C01778=1014.459,160.454,-126.016,166.827,55.652,160.236
C01779=1014.455,160.205,-125.996,166.824,55.663,160.237
C01780=1014.451,159.957,-125.976,166.820,55.675,160.239
C01781=1014.447,159.707,-125.956,166.816,55.686,160.240
C01782=1014.443,159.458,-125.936,166.813,55.697,160.242
C01783=1014.439,159.209,-125.916,166.809,55.709,160.243
C01784=1014.435,158.960,-125.897,166.807,55.720,160.245
C01785=1014.431,158.710,-125.877,166.803,55.731,160.246
C01786=1014.428,158.461,-125.856,166.799,55.742,160.248
C01787=1014.423,158.212,-125.837,166.796,55.754,160.249
C01788=1014.419,157.963,-125.818,166.792,55.765,160.250
C01789=1014.415,157.714,-125.798,166.788,55.776,160.252
C01790=1014.411,157.464,-125.779,166.785,55.788,160.253
C01791=1014.406,157.215,-125.760,166.781,55.799,160.255
C01792=1014.403,156.966,-125.740,166.778,55.811,160.256
C01793=1014.398,156.716,-125.720,166.774,55.823,160.258
C01794=1014.393,156.467,-125.700,166.771,55.834,160.259
C01795=1014.389,156.217,-125.682,166.767,55.846,160.261
C01796=1014.385,155.968,-125.662,166.763,55.857,160.262
C01797=1014.381,155.719,-125.643,166.760,55.868,160.264
C01798=1014.376,155.470,-125.623,166.756,55.880,160.265
C01799=1014.372,155.221,-125.605,166.753,55.891,160.267
C01800=1014.367,154.941,-125.582,166.749,55.904,160.268
C01801=1014.363,154.661,-125.561,166.745,55.917,160.270
C01802=1014.358,154.381,-125.539,166.741,55.930,160.272
C01803=1014.354,154.101,-125.517,166.737,55.943,160.273
C01804=1014.350,153.852,-125.498,166.733,55.954,160.275
C01805=1014.345,153.602,-125.479,166.731,55.965,160.276
C01806=1014.341,153.353,-125.459,166.728,55.977,160.278
C01807=1014.337,153.104,-125.440,166.724,55.989,160.279
C01808=1014.333,152.855,-125.421,166.721,56.000,160.281
C01809=1014.328,152.606,-125.401,166.717,56.011,160.282
C01810=1014.324,152.356,-125.383,166.713,56.023,160.284
C01811=1014.320,152.108,-125.364,166.710,56.034,160.285
C01812=1014.316,151.858,-125.345,166.706,56.046,160.287
C01813=1014.312,151.609,-125.325,166.703,56.058,160.288
C01814=1014.308,151.360,-125.306,166.700,56.069,160.290
C01815=1014.304,151.110,-125.287,166.697,56.080,160.291
C01816=1014.299,150.861,-125.268,166.693,56.091,160.293
C01817=1014.295,150.612,-125.249,166.690,56.103,160.294
C01818=1014.291,150.363,-125.229,166.686,56.115,160.296
C01819=1014.287,150.113,-125.211,166.683,56.126,160.297
C01820=1014.283,149.864,-125.191,166.680,56.138,160.299
C01821=1014.279,149.615,-125.173,166.676,56.149,160.300
C01822=1014.275,149.366,-125.153,166.673,56.160,160.302
C01823=1014.270,149.116,-125.135,166.670,56.172,160.303
C01824=1014.266,148.867,-125.116,166.667,56.183,160.305
C01825=1014.262,148.618,-125.097,166.663,56.194,160.306
C01826=1014.257,148.369,-125.077,166.659,56.206,160.308
C01827=1014.253,148.119,-125.059,166.656,56.218,160.309
C01828=1014.249,147.870,-125.039,166.654,56.229,160.311
C01829=1014.245,147.621,-125.021,166.650,56.240,160.312
C01830=1014.241,147.372,-125.001,166.646,56.252,160.314
C01831=1014.237,147.122,-124.983,166.643,56.263,160.315
C01832=1014.233,146.873,-124.964,166.640,56.275,160.317
C01833=1014.229,146.624,-124.944,166.636,56.286,160.318
C01834=1014.224,146.374,-124.926,166.633,56.297,160.320
C01835=1014.220,146.126,-124.907,166.630,56.309,160.321
C01836=1014.216,145.876,-124.888,166.627,56.321,160.323
C01837=1014.212,145.627,-124.870,166.623,56.332,160.324
C01838=1014.208,145.378,-124.850,166.620,56.343,160.326
C01839=1014.204,145.128,-124.831,166.617,56.355,160.327
C01840=1014.199,144.879,-124.814,166.614,56.366,160.329
C01841=1014.195,144.630,-124.795,166.610,56.378,160.330
C01842=1014.191,144.381,-124.775,166.607,56.389,160.332
C01843=1014.186,144.131,-124.757,166.603,56.401,160.333
C01844=1014.182,143.882,-124.738,166.601,56.412,160.335
C01845=1014.178,143.633,-124.721,166.598,56.424,160.336
C01846=1014.174,143.384,-124.701,166.594,56.435,160.338
C01847=1014.170,143.134,-124.682,166.591,56.446,160.339
C01848=1014.165,142.885,-124.664,166.587,56.458,160.341
C01849=1014.161,142.636,-124.646,166.585,56.469,160.342
C01850=1014.157,142.386,-124.627,166.582,56.481,160.344
C01851=1014.153,142.137,-124.609,166.578,56.492,160.345
C01852=1014.148,141.888,-124.589,166.575,56.504,160.347
C01853=1014.145,141.639,-124.571,166.572,56.515,160.349
C01854=1014.140,141.390,-124.553,166.568,56.526,160.350
C01855=1014.136,141.140,-124.534,166.565,56.538,160.351
C01856=1014.132,140.890,-124.515,166.562,56.550,160.353
C01857=1014.128,140.642,-124.498,166.560,56.561,160.355
C01858=1014.124,140.392,-124.479,166.556,56.572,160.356
C01859=1014.119,140.143,-124.459,166.553,56.584,160.357
C01860=1014.115,139.894,-124.442,166.550,56.595,160.359
C01861=1014.111,139.645,-124.423,166.546,56.606,160.360
C01862=1014.107,139.395,-124.404,166.543,56.618,160.362
C01863=1014.102,139.146,-124.386,166.540,56.629,160.364
C01864=1014.098,138.866,-124.365,166.537,56.642,160.365
C01865=1014.094,138.586,-124.344,166.533,56.654,160.367
C01866=1014.088,138.306,-124.323,166.529,56.667,160.368
C01867=1014.085,138.026,-124.303,166.526,56.680,160.370
C01868=1014.080,137.776,-124.285,166.523,56.691,160.372
C01869=1014.076,137.527,-124.266,166.520,56.703,160.373
C01870=1014.072,137.278,-124.248,166.516,56.714,160.375
C01871=1014.068,137.028,-124.230,166.514,56.725,160.376
C01872=1014.063,136.779,-124.211,166.511,56.737,160.378
C01873=1014.060,136.530,-124.193,166.507,56.748,160.379
C01874=1014.055,136.281,-124.175,166.505,56.759,160.381
C01875=1014.051,136.031,-124.156,166.502,56.771,160.383
C01876=1014.047,135.782,-124.138,166.498,56.782,160.384
C01877=1014.043,135.533,-124.119,166.496,56.794,160.386
C01878=1014.038,135.283,-124.101,166.493,56.805,160.387
C01879=1014.034,135.034,-124.083,166.489,56.817,160.388
C01880=1014.030,134.784,-124.065,166.487,56.828,160.390
C01881=1014.025,134.535,-124.047,166.483,56.839,160.391
C01882=1014.022,134.286,-124.029,166.480,56.851,160.393
C01883=1014.017,134.037,-124.011,166.478,56.862,160.395
C01884=1014.013,133.788,-123.993,166.474,56.873,160.396
C01885=1014.009,133.538,-123.974,166.471,56.885,160.398
C01886=1014.004,133.288,-123.957,166.469,56.896,160.399
C01887=1014.001,133.039,-123.938,166.465,56.907,160.401
C01888=1013.996,132.790,-123.920,166.463,56.919,160.402
C01889=1013.992,132.541,-123.902,166.459,56.930,160.404
C01890=1013.988,132.291,-123.884,166.456,56.942,160.405
C01891=1013.984,132.043,-123.867,166.454,56.953,160.407
C01892=1013.979,131.793,-123.848,166.450,56.964,160.408
C01893=1013.975,131.544,-123.830,166.448,56.975,160.410
C01894=1013.971,131.295,-123.812,166.444,56.987,160.411
C01895=1013.967,131.045,-123.794,166.441,56.998,160.413
C01896=1013.963,130.796,-123.776,166.438,57.009,160.414
C01897=1013.958,130.547,-123.758,166.435,57.021,160.416
C01898=1013.955,130.298,-123.739,166.432,57.032,160.418
C01899=1013.950,130.048,-123.722,166.429,57.043,160.419
C01900=1013.946,129.798,-123.703,166.427,57.054,160.421
C01901=1013.942,129.549,-123.685,166.424,57.066,160.422
C01902=1013.938,129.299,-123.668,166.421,57.077,160.424
C01903=1013.933,129.051,-123.650,166.418,57.088,160.425
C01904=1013.929,128.801,-123.633,166.415,57.100,160.427
C01905=1013.925,128.552,-123.615,166.412,57.111,160.428
C01906=1013.921,128.302,-123.597,166.409,57.123,160.430
C01907=1013.917,128.053,-123.579,166.406,57.135,160.431
C01908=1013.912,127.803,-123.562,166.403,57.145,160.433
C01909=1013.908,127.555,-123.544,166.400,57.157,160.435
C01910=1013.904,127.305,-123.526,166.397,57.168,160.436
C01911=1013.899,127.056,-123.509,166.394,57.180,160.438
C01912=1013.895,126.806,-123.491,166.391,57.192,160.439
C01913=1013.891,126.557,-123.474,166.389,57.202,160.441
C01914=1013.886,126.307,-123.456,166.386,57.214,160.442
C01915=1013.882,126.058,-123.439,166.383,57.225,160.444
C01916=1013.878,125.809,-123.421,166.380,57.237,160.445
C01917=1013.874,125.559,-123.404,166.377,57.247,160.447
C01918=1013.869,125.310,-123.386,166.374,57.259,160.448
C01919=1013.865,125.061,-123.368,166.371,57.270,160.450
C01920=1013.861,124.811,-123.351,166.369,57.282,160.452
C01921=1013.856,124.562,-123.333,166.366,57.294,160.453
C01922=1013.852,124.312,-123.316,166.363,57.304,160.455
C01923=1013.848,124.064,-123.298,166.360,57.316,160.456
C01924=1013.843,123.814,-123.281,166.357,57.327,160.458
C01925=1013.839,123.564,-123.263,166.354,57.338,160.459
C01926=1013.835,123.315,-123.245,166.352,57.350,160.461
C01927=1013.831,123.066,-123.228,166.348,57.361,160.462
C01928=1013.826,122.786,-123.209,166.346,57.373,160.464
C01929=1013.821,122.506,-123.189,166.342,57.386,160.466
C01930=1013.817,122.226,-123.169,166.340,57.399,160.468
C01931=1013.812,121.946,-123.150,166.336,57.411,160.469
C01932=1013.807,121.697,-123.132,166.334,57.423,160.471
C01933=1013.803,121.447,-123.115,166.330,57.434,160.472
C01934=1013.799,121.197,-123.097,166.328,57.445,160.474
C01935=1013.795,120.949,-123.080,166.326,57.456,160.475
C01936=1013.791,120.699,-123.063,166.322,57.467,160.477
C01937=1013.786,120.449,-123.045,166.319,57.478,160.478
C01938=1013.782,120.201,-123.027,166.316,57.490,160.480
C01939=1013.778,119.952,-123.010,166.314,57.501,160.481
C01940=1013.774,119.702,-122.993,166.311,57.511,160.483
C01941=1013.770,119.453,-122.975,166.308,57.523,160.485
C01942=1013.765,119.203,-122.958,166.306,57.534,160.486
C01943=1013.761,118.954,-122.940,166.302,57.545,160.487
C01944=1013.757,118.704,-122.923,166.300,57.557,160.489
C01945=1013.753,118.455,-122.905,166.298,57.568,160.491
C01946=1013.749,118.206,-122.888,166.294,57.579,160.492
C01947=1013.745,117.956,-122.871,166.292,57.589,160.493
C01948=1013.740,117.707,-122.854,166.290,57.601,160.495
C01949=1013.736,117.458,-122.836,166.286,57.612,160.497
C01950=1013.732,117.209,-122.819,166.284,57.623,160.498
C01951=1013.728,116.959,-122.801,166.281,57.634,160.500
C01952=1013.724,116.709,-122.784,166.279,57.645,160.501
C01953=1013.720,116.461,-122.766,166.276,57.656,160.503
C01954=1013.715,116.211,-122.749,166.273,57.667,160.504
C01955=1013.712,115.961,-122.731,166.271,57.678,160.506
C01956=1013.708,115.712,-122.714,166.267,57.689,160.507
C01957=1013.704,115.462,-122.697,166.265,57.700,160.509
C01958=1013.700,115.213,-122.679,166.263,57.711,160.510
C01959=1013.696,114.964,-122.662,166.261,57.722,160.512
C01960=1013.691,114.714,-122.644,166.257,57.733,160.513
C01961=1013.687,114.465,-122.627,166.255,57.744,160.515
C01962=1013.683,114.215,-122.610,166.252,57.755,160.516
C01963=1013.680,113.966,-122.593,166.250,57.766,160.518
C01964=1013.675,113.717,-122.575,166.247,57.777,160.519
C01965=1013.671,113.468,-122.558,166.244,57.788,160.521
C01966=1013.667,113.218,-122.541,166.241,57.799,160.522
C01967=1013.663,112.969,-122.524,166.239,57.809,160.524
C01968=1013.659,112.719,-122.506,166.237,57.821,160.526
C01969=1013.655,112.470,-122.489,166.235,57.832,160.527
C01970=1013.651,112.221,-122.472,166.232,57.843,160.529
C01971=1013.647,111.972,-122.454,166.229,57.854,160.530
C01972=1013.642,111.722,-122.437,166.226,57.865,160.532
C01973=1013.638,111.473,-122.421,166.224,57.875,160.533
C01974=1013.634,111.224,-122.403,166.221,57.886,160.535
C01975=1013.630,110.973,-122.387,166.218,57.897,160.536
C01976=1013.625,110.724,-122.370,166.215,57.908,160.537
C01977=1013.621,110.475,-122.353,166.213,57.919,160.539
C01978=1013.617,110.226,-122.336,166.211,57.930,160.541
C01979=1013.613,109.977,-122.320,166.208,57.941,160.542
C01980=1013.608,109.727,-122.302,166.205,57.953,160.544
C01981=1013.604,109.477,-122.285,166.203,57.964,160.545
C01982=1013.600,109.228,-122.268,166.201,57.974,160.547
C01983=1013.596,108.979,-122.251,166.198,57.985,160.548
C01984=1013.591,108.729,-122.234,166.196,57.996,160.550
C01985=1013.587,108.480,-122.218,166.192,58.007,160.551
C01986=1013.583,108.230,-122.201,166.190,58.018,160.553
C01987=1013.579,107.981,-122.185,166.188,58.029,160.554
C01988=1013.575,107.732,-122.168,166.185,58.040,160.556
C01989=1013.570,107.482,-122.151,166.183,58.051,160.557
C01990=1013.566,107.233,-122.134,166.179,58.062,160.559
C01991=1013.561,106.984,-122.118,166.177,58.073,160.560
C01992=1013.557,106.704,-122.099,166.175,58.085,160.562
C01993=1013.552,106.423,-122.081,166.172,58.097,160.564
C01994=1013.547,106.144,-122.061,166.169,58.109,160.566
C01995=1013.542,105.864,-122.043,166.166,58.121,160.567
C01996=1013.538,105.615,-122.026,166.163,58.133,160.569
C01997=1013.534,105.365,-122.010,166.161,58.144,160.570
C01998=1013.530,105.116,-121.993,166.158,58.154,160.572
C01999=1013.525,104.867,-121.976,166.156,58.165,160.573
C02000=1013.522,104.617,-121.960,166.154,58.176,160.575
C02001=1013.517,104.367,-121.943,166.151,58.187,160.576
C02002=1013.513,104.118,-121.926,166.149,58.198,160.578
C02003=1013.508,103.869,-121.910,166.147,58.209,160.579
C02004=1013.505,103.619,-121.893,166.144,58.220,160.581
C02005=1013.500,103.370,-121.877,166.141,58.231,160.582
C02006=1013.496,103.121,-121.860,166.139,58.242,160.584
C02007=1013.492,102.871,-121.844,166.136,58.253,160.586
C02008=1013.488,102.622,-121.827,166.133,58.263,160.587
C02009=1013.483,102.372,-121.811,166.131,58.274,160.588
C02010=1013.479,102.123,-121.794,166.129,58.285,160.590
C02011=1013.475,101.874,-121.777,166.126,58.295,160.591
C02012=1013.471,101.624,-121.761,166.124,58.306,160.593
C02013=1013.467,101.374,-121.744,166.122,58.317,160.595
C02014=1013.463,101.125,-121.727,166.119,58.327,160.596
C02015=1013.459,100.876,-121.711,166.117,58.338,160.597
C02016=1013.454,100.627,-121.694,166.114,58.349,160.599
C02017=1013.450,100.377,-121.677,166.112,58.360,160.601
C02018=1013.446,100.128,-121.662,166.109,58.370,160.602
C02019=1013.442,99.878,-121.644,166.107,58.381,160.603
C02020=1013.437,99.628,-121.628,166.106,58.391,160.605
C02021=1013.434,99.379,-121.611,166.103,58.402,160.607
C02022=1013.429,99.130,-121.595,166.100,58.412,160.608
C02023=1013.425,98.880,-121.578,166.098,58.423,160.610
C02024=1013.421,98.631,-121.562,166.096,58.434,160.611
C02025=1013.416,98.382,-121.546,166.093,58.444,160.612
C02026=1013.412,98.132,-121.530,166.091,58.455,160.614
C02027=1013.408,97.883,-121.513,166.088,58.466,160.616
C02028=1013.404,97.633,-121.498,166.086,58.477,160.617
C02029=1013.399,97.384,-121.481,166.084,58.488,160.619
C02030=1013.395,97.135,-121.465,166.081,58.498,160.620
C02031=1013.391,96.885,-121.449,166.079,58.509,160.622
C02032=1013.387,96.636,-121.432,166.077,58.520,160.623
C02033=1013.383,96.386,-121.417,166.074,58.530,160.624
C02034=1013.378,96.137,-121.401,166.072,58.541,160.626
C02035=1013.374,95.888,-121.384,166.069,58.552,160.628
C02036=1013.370,95.638,-121.368,166.067,58.563,160.629
C02037=1013.366,95.388,-121.352,166.064,58.573,160.630
C02038=1013.361,95.139,-121.336,166.062,58.584,160.632
C02039=1013.357,94.890,-121.320,166.059,58.594,160.633
C02040=1013.353,94.640,-121.304,166.058,58.605,160.635
C02041=1013.349,94.391,-121.287,166.056,58.616,160.637
C02042=1013.344,94.141,-121.271,166.053,58.626,160.638
C02043=1013.340,93.892,-121.256,166.051,58.637,160.639
C02044=1013.335,93.643,-121.239,166.048,58.647,160.641
C02045=1013.331,93.393,-121.223,166.046,58.658,160.642
C02046=1013.328,93.143,-121.207,166.043,58.669,160.644
C02047=1013.323,92.894,-121.191,166.042,58.679,160.645
C02048=1013.319,92.645,-121.175,166.040,58.689,160.647
C02049=1013.314,92.395,-121.159,166.037,58.700,160.648
C02050=1013.310,92.146,-121.143,166.035,58.711,160.650
C02051=1013.306,91.896,-121.126,166.032,58.721,160.651
C02052=1013.302,91.647,-121.110,166.031,58.731,160.653
C02053=1013.298,91.397,-121.095,166.028,58.742,160.654
C02054=1013.293,91.148,-121.078,166.025,58.752,160.655
C02055=1013.289,90.899,-121.062,166.023,58.763,160.657
C02056=1013.285,90.619,-121.044,166.021,58.774,160.659
C02057=1013.279,90.339,-121.026,166.018,58.786,160.660
C02058=1013.275,90.060,-121.008,166.015,58.798,160.662
C02059=1013.270,89.781,-120.990,166.013,58.809,160.664
C02060=1013.266,89.531,-120.975,166.011,58.819,160.665
C02061=1013.262,89.282,-120.958,166.008,58.830,160.667
C02062=1013.258,89.032,-120.942,166.007,58.840,160.668
C02063=1013.254,88.782,-120.927,166.004,58.850,160.669
C02064=1013.249,88.533,-120.910,166.002,58.861,160.671
C02065=1013.245,88.284,-120.894,166.000,58.871,160.673
C02066=1013.240,88.034,-120.879,165.998,58.882,160.674
C02067=1013.236,87.785,-120.863,165.995,58.892,160.675
C02068=1013.232,87.535,-120.847,165.992,58.902,160.677
C02069=1013.227,87.286,-120.831,165.991,58.913,160.679
C02070=1013.223,87.036,-120.816,165.989,58.923,160.680
C02071=1013.219,86.787,-120.800,165.986,58.934,160.681
C02072=1013.214,86.538,-120.785,165.984,58.944,160.683
C02073=1013.210,86.288,-120.769,165.982,58.954,160.684
C02074=1013.206,86.039,-120.753,165.980,58.965,160.686
C02075=1013.201,85.789,-120.738,165.977,58.975,160.687
C02076=1013.197,85.539,-120.722,165.975,58.985,160.689
C02077=1013.193,85.290,-120.706,165.973,58.996,160.690
C02078=1013.189,85.040,-120.691,165.971,59.006,160.692
C02079=1013.185,84.790,-120.675,165.969,59.016,160.693
C02080=1013.180,84.542,-120.660,165.966,59.026,160.694
C02081=1013.176,84.292,-120.645,165.964,59.037,160.696
C02082=1013.172,84.042,-120.629,165.962,59.047,160.697
C02083=1013.167,83.793,-120.613,165.960,59.057,160.699
C02084=1013.163,83.543,-120.597,165.958,59.067,160.700
C02085=1013.159,83.294,-120.582,165.955,59.077,160.702
C02086=1013.154,83.044,-120.566,165.954,59.087,160.703
C02087=1013.151,82.795,-120.550,165.952,59.098,160.705
C02088=1013.146,82.546,-120.535,165.949,59.108,160.706
C02089=1013.141,82.296,-120.520,165.947,59.118,160.708
C02090=1013.137,82.047,-120.504,165.945,59.128,160.709
C02091=1013.133,81.797,-120.488,165.943,59.138,160.710
C02092=1013.129,81.548,-120.473,165.940,59.149,160.712
C02093=1013.125,81.298,-120.458,165.939,59.158,160.713
C02094=1013.121,81.049,-120.442,165.936,59.169,160.714
C02095=1013.116,80.799,-120.426,165.934,59.178,160.716
C02096=1013.111,80.550,-120.411,165.932,59.189,160.717
C02097=1013.107,80.300,-120.395,165.930,59.199,160.719
C02098=1013.103,80.051,-120.380,165.927,59.209,160.720
C02099=1013.099,79.802,-120.364,165.926,59.219,160.722
C02100=1013.095,79.551,-120.349,165.923,59.229,160.723
C02101=1013.091,79.302,-120.333,165.921,59.239,160.724
C02102=1013.086,79.052,-120.317,165.920,59.249,160.726
C02103=1013.083,78.803,-120.302,165.917,59.259,160.727
C02104=1013.078,78.554,-120.287,165.915,59.269,160.729
C02105=1013.073,78.305,-120.271,165.913,59.279,160.730
C02106=1013.069,78.055,-120.255,165.911,59.289,160.732
C02107=1013.066,77.806,-120.240,165.910,59.299,160.733
C02108=1013.061,77.556,-120.225,165.906,59.308,160.734
C02109=1013.057,77.306,-120.209,165.905,59.318,160.736
C02110=1013.053,77.057,-120.193,165.903,59.328,160.737
C02111=1013.049,76.807,-120.178,165.900,59.338,160.739
C02112=1013.044,76.558,-120.163,165.899,59.348,160.740
C02113=1013.040,76.308,-120.148,165.897,59.358,160.742
C02114=1013.036,76.059,-120.132,165.894,59.367,160.743
C02115=1013.031,75.809,-120.117,165.892,59.377,160.744
C02116=1013.027,75.560,-120.102,165.891,59.387,160.746
C02117=1013.023,75.311,-120.086,165.888,59.397,160.747
C02118=1013.018,75.061,-120.072,165.887,59.407,160.749
C02119=1013.014,74.811,-120.056,165.884,59.418,160.750
C02120=1013.010,74.572,-120.042,165.882,59.427,160.751
C02121=1013.006,74.331,-120.027,165.880,59.436,160.752
C02122=1013.002,74.092,-120.013,165.878,59.446,160.754
C02123=1012.997,73.852,-119.998,165.876,59.455,160.755
C02124=1012.994,73.612,-119.983,165.874,59.465,160.757
C02125=1012.989,73.372,-119.969,165.872,59.474,160.758
C02126=1012.985,73.133,-119.955,165.870,59.484,160.759
C02127=1012.981,72.892,-119.940,165.868,59.493,160.761
C02128=1012.977,72.643,-119.925,165.867,59.503,160.762
C02129=1012.973,72.393,-119.910,165.865,59.512,160.763
C02130=1012.968,72.144,-119.895,165.862,59.522,160.765
C02131=1012.964,71.895,-119.879,165.860,59.532,160.766
C02132=1012.959,71.645,-119.865,165.858,59.541,160.767
C02133=1012.955,71.396,-119.849,165.857,59.551,160.769
C02134=1012.951,71.147,-119.835,165.854,59.560,160.770
C02135=1012.947,70.897,-119.819,165.852,59.570,160.771
C02136=1012.943,70.647,-119.804,165.850,59.580,160.773
C02137=1012.938,70.398,-119.789,165.848,59.589,160.774
C02138=1012.934,70.148,-119.774,165.847,59.599,160.776
C02139=1012.929,69.899,-119.759,165.844,59.608,160.777
C02140=1012.926,69.649,-119.744,165.843,59.618,160.779
C02141=1012.921,69.400,-119.729,165.840,59.628,160.780
C02142=1012.917,69.150,-119.714,165.838,59.638,160.781
C02143=1012.912,68.901,-119.699,165.836,59.647,160.782
C02144=1012.908,68.651,-119.684,165.835,59.657,160.784
C02145=1012.903,68.402,-119.669,165.832,59.666,160.785
C02146=1012.900,68.152,-119.654,165.830,59.675,160.786
C02147=1012.895,67.903,-119.639,165.829,59.685,160.788
C02148=1012.891,67.653,-119.624,165.827,59.694,160.789
C02149=1012.887,67.404,-119.610,165.825,59.704,160.791
C02150=1012.882,67.154,-119.594,165.823,59.713,160.792
C02151=1012.878,66.904,-119.580,165.821,59.723,160.793
C02152=1012.874,66.655,-119.565,165.818,59.733,160.794
C02153=1012.869,66.405,-119.550,165.816,59.742,160.796
C02154=1012.865,66.156,-119.536,165.815,59.752,160.797
C02155=1012.861,65.906,-119.521,165.812,59.761,160.798
C02156=1012.856,65.657,-119.506,165.810,59.770,160.800
C02157=1012.853,65.407,-119.491,165.809,59.780,160.801
C02158=1012.848,65.157,-119.477,165.807,59.789,160.802
C02159=1012.843,64.909,-119.462,165.805,59.798,160.804
C02160=1012.839,64.659,-119.447,165.803,59.808,160.805
C02161=1012.835,64.409,-119.432,165.801,59.817,160.806
C02162=1012.830,64.160,-119.417,165.799,59.826,160.808
C02163=1012.826,63.910,-119.402,165.797,59.836,160.809
C02164=1012.822,63.661,-119.388,165.795,59.845,160.811
C02165=1012.817,63.411,-119.374,165.793,59.855,160.812
C02166=1012.813,63.161,-119.358,165.791,59.864,160.813
C02167=1012.809,62.912,-119.344,165.790,59.873,160.814
C02168=1012.804,62.662,-119.329,165.788,59.882,160.816
C02169=1012.801,62.413,-119.315,165.786,59.891,160.817
C02170=1012.796,62.163,-119.300,165.784,59.901,160.818
C02171=1012.791,61.913,-119.286,165.782,59.910,160.820
C02172=1012.787,61.664,-119.272,165.780,59.919,160.821
C02173=1012.782,61.414,-119.257,165.778,59.928,160.822
C02174=1012.778,61.165,-119.243,165.777,59.938,160.824
C02175=1012.773,60.915,-119.228,165.775,59.947,160.825
C02176=1012.769,60.666,-119.214,165.773,59.957,160.826
C02177=1012.764,60.416,-119.200,165.770,59.966,160.827
C02178=1012.760,60.167,-119.185,165.768,59.975,160.829
C02179=1012.755,59.917,-119.171,165.766,59.984,160.830
C02180=1012.732,71.816,-120.285,165.827,59.747,160.800
C02181=1012.736,72.066,-120.299,165.829,59.737,160.799
C02182=1012.741,72.316,-120.315,165.831,59.728,160.797
C02183=1012.745,72.565,-120.329,165.833,59.719,160.796
C02184=1012.749,72.814,-120.345,165.834,59.709,160.795
C02185=1012.753,73.059,-120.359,165.837,59.700,160.793
C02186=1012.757,73.305,-120.373,165.839,59.691,160.792
C02187=1012.762,73.551,-120.388,165.840,59.681,160.791
C02188=1012.765,73.796,-120.403,165.842,59.672,160.789
C02189=1012.770,74.042,-120.418,165.844,59.662,160.788
C02190=1012.774,74.286,-120.433,165.846,59.653,160.787
C02191=1012.778,74.532,-120.448,165.848,59.644,160.785
C02192=1012.783,74.778,-120.463,165.851,59.633,160.784
C02193=1012.787,75.026,-120.478,165.853,59.624,160.783
C02194=1012.791,75.276,-120.493,165.854,59.614,160.781
C02195=1012.796,75.526,-120.508,165.856,59.604,160.780
C02196=1012.799,75.775,-120.523,165.858,59.595,160.778
C02197=1012.803,76.025,-120.539,165.861,59.585,160.777
C02198=1012.809,76.274,-120.554,165.863,59.576,160.776
C02199=1012.812,76.524,-120.569,165.864,59.566,160.774
C02200=1012.816,76.773,-120.584,165.866,59.556,160.773
C02201=1012.820,77.024,-120.599,165.868,59.547,160.772
C02202=1012.825,77.273,-120.615,165.871,59.537,160.770
C02203=1012.829,77.522,-120.630,165.873,59.528,160.769
C02204=1012.833,77.771,-120.646,165.874,59.518,160.767
C02205=1012.837,78.021,-120.661,165.876,59.508,160.766
C02206=1012.842,78.271,-120.677,165.879,59.498,160.765
C02207=1012.845,78.520,-120.692,165.881,59.488,160.763
C02208=1012.850,78.769,-120.708,165.882,59.478,160.762
C02209=1012.854,79.020,-120.723,165.884,59.469,160.761
C02210=1012.858,79.268,-120.738,165.887,59.459,160.759
C02211=1012.862,79.518,-120.753,165.889,59.449,160.758
C02212=1012.867,79.767,-120.769,165.890,59.439,160.756
C02213=1012.871,80.017,-120.785,165.894,59.430,160.755
C02214=1012.874,80.266,-120.800,165.895,59.420,160.754
C02215=1012.879,80.516,-120.815,165.897,59.410,160.752
C02216=1012.883,80.766,-120.831,165.899,59.400,160.751
C02217=1012.887,81.015,-120.847,165.901,59.390,160.749
C02218=1012.891,81.264,-120.862,165.902,59.380,160.748
C02219=1012.896,81.513,-120.878,165.906,59.371,160.747
C02220=1012.900,81.764,-120.893,165.907,59.361,160.745
C02221=1012.904,82.013,-120.908,165.910,59.350,160.744
C02222=1012.908,82.262,-120.924,165.911,59.341,160.742
C02223=1012.912,82.512,-120.940,165.913,59.331,160.741
C02224=1012.917,82.761,-120.955,165.916,59.320,160.740
C02225=1012.921,83.011,-120.971,165.917,59.311,160.738
C02226=1012.925,83.261,-120.986,165.920,59.300,160.737
C02227=1012.929,83.509,-121.001,165.922,59.290,160.735
C02228=1012.934,83.759,-121.017,165.924,59.280,160.734
C02229=1012.938,84.009,-121.032,165.926,59.270,160.732
C02230=1012.942,84.258,-121.048,165.928,59.260,160.731
C02231=1012.947,84.508,-121.064,165.930,59.250,160.729
C02232=1012.950,84.757,-121.079,165.933,59.240,160.728
C02233=1012.954,85.007,-121.094,165.934,59.230,160.727
C02234=1012.959,85.256,-121.110,165.937,59.220,160.725
C02235=1012.964,85.506,-121.125,165.939,59.210,160.724
C02236=1012.968,85.755,-121.141,165.941,59.200,160.722
C02237=1012.972,86.005,-121.157,165.942,59.189,160.721
C02238=1012.976,86.254,-121.172,165.945,59.179,160.719
C02239=1012.980,86.503,-121.188,165.948,59.169,160.718
C02240=1012.985,86.753,-121.204,165.949,59.159,160.716
C02241=1012.989,87.002,-121.220,165.952,59.149,160.715
C02242=1012.993,87.252,-121.235,165.954,59.139,160.714
C02243=1012.997,87.502,-121.251,165.956,59.128,160.712
C02244=1013.002,87.750,-121.266,165.958,59.117,160.711
C02245=1013.006,88.000,-121.282,165.960,59.108,160.709
C02246=1013.010,88.250,-121.297,165.963,59.097,160.708
C02247=1013.015,88.500,-121.313,165.965,59.086,160.706
C02248=1013.019,88.749,-121.328,165.966,59.077,160.705
C02249=1013.023,88.998,-121.345,165.969,59.066,160.703
C02250=1013.027,89.248,-121.361,165.972,59.056,160.702
C02251=1013.031,89.498,-121.377,165.974,59.046,160.701
C02252=1013.035,89.746,-121.392,165.976,59.035,160.699
C02253=1013.041,90.026,-121.410,165.978,59.024,160.697
C02254=1013.045,90.306,-121.429,165.981,59.013,160.696
C02255=1013.049,90.585,-121.446,165.982,59.001,160.694
C02256=1013.054,90.864,-121.464,165.986,58.990,160.693
C02257=1013.058,91.114,-121.480,165.988,58.979,160.691
C02258=1013.062,91.363,-121.496,165.989,58.969,160.689
C02259=1013.067,91.613,-121.512,165.992,58.959,160.688
C02260=1013.070,91.862,-121.529,165.995,58.948,160.687
C02261=1013.075,92.112,-121.545,165.996,58.938,160.685
C02262=1013.078,92.360,-121.560,165.999,58.928,160.684
C02263=1013.083,92.610,-121.576,166.001,58.917,160.682
C02264=1013.087,92.860,-121.592,166.004,58.906,160.681
C02265=1013.091,93.109,-121.609,166.005,58.897,160.679
C02266=1013.095,93.358,-121.624,166.008,58.886,160.678
C02267=1013.100,93.608,-121.640,166.010,58.876,160.676
C02268=1013.104,93.858,-121.656,166.013,58.865,160.675
C02269=1013.108,94.107,-121.672,166.014,58.855,160.673
C02270=1013.112,94.356,-121.689,166.017,58.845,160.672
C02271=1013.116,94.606,-121.705,166.019,58.834,160.670
C02272=1013.121,94.856,-121.720,166.022,58.823,160.669
C02273=1013.125,95.105,-121.737,166.024,58.812,160.668
C02274=1013.130,95.354,-121.753,166.026,58.803,160.666
C02275=1013.133,95.604,-121.769,166.028,58.792,160.664
C02276=1013.137,95.854,-121.785,166.030,58.781,160.663
C02277=1013.142,96.103,-121.801,166.033,58.771,160.662
C02278=1013.146,96.352,-121.817,166.035,58.760,160.660
C02279=1013.151,96.602,-121.833,166.038,58.749,160.659
C02280=1013.154,96.850,-121.849,166.040,58.739,160.657
C02281=1013.158,97.100,-121.865,166.042,58.729,160.656
C02282=1013.163,97.349,-121.881,166.044,58.718,160.654
C02283=1013.167,97.599,-121.897,166.047,58.708,160.653
C02284=1013.171,97.848,-121.913,166.049,58.697,160.651
C02285=1013.175,98.098,-121.930,166.051,58.686,160.650
C02286=1013.179,98.347,-121.945,166.054,58.675,160.648
C02287=1013.184,98.596,-121.962,166.056,58.665,160.647
C02288=1013.187,98.846,-121.978,166.058,58.654,160.645
C02289=1013.193,99.096,-121.995,166.061,58.643,160.644
C02290=1013.196,99.346,-122.011,166.063,58.632,160.642
C02291=1013.201,99.595,-122.028,166.066,58.622,160.641
C02292=1013.204,99.845,-122.044,166.067,58.612,160.639
C02293=1013.209,100.094,-122.061,166.069,58.601,160.638
C02294=1013.213,100.344,-122.077,166.072,58.591,160.636
C02295=1013.217,100.592,-122.094,166.074,58.580,160.635
C02296=1013.221,100.842,-122.110,166.077,58.570,160.633
C02297=1013.225,101.091,-122.126,166.079,58.559,160.632
C02298=1013.229,101.341,-122.143,166.082,58.548,160.630
C02299=1013.234,101.590,-122.159,166.084,58.537,160.629
C02300=1013.237,101.839,-122.176,166.087,58.527,160.627
C02301=1013.242,102.089,-122.192,166.089,58.516,160.626
C02302=1013.246,102.338,-122.209,166.091,58.505,160.624
C02303=1013.250,102.588,-122.225,166.094,58.495,160.623
C02304=1013.254,102.837,-122.242,166.096,58.484,160.621
C02305=1013.258,103.087,-122.258,166.099,58.473,160.620
C02306=1013.262,103.336,-122.275,166.101,58.462,160.618
C02307=1013.267,103.585,-122.291,166.104,58.452,160.617
C02308=1013.270,103.835,-122.308,166.106,58.441,160.615
C02309=1013.275,104.084,-122.324,166.108,58.430,160.614
C02310=1013.278,104.334,-122.341,166.111,58.419,160.612
C02311=1013.284,104.583,-122.357,166.113,58.408,160.611
C02312=1013.287,104.833,-122.375,166.115,58.397,160.609
C02313=1013.292,105.082,-122.390,166.118,58.387,160.608
C02314=1013.296,105.331,-122.407,166.120,58.376,160.606
C02315=1013.300,105.580,-122.424,166.123,58.365,160.605
C02316=1013.304,105.830,-122.440,166.125,58.355,160.603
C02317=1013.309,106.110,-122.460,166.129,58.342,160.602
C02318=1013.314,106.390,-122.478,166.131,58.330,160.600
C02319=1013.318,106.669,-122.496,166.133,58.317,160.598
C02320=1013.323,106.949,-122.514,166.136,58.305,160.596
C02321=1013.327,107.198,-122.531,166.138,58.294,160.595
C02322=1013.332,107.447,-122.548,166.141,58.283,160.593
C02323=1013.335,107.697,-122.564,166.143,58.273,160.592
C02324=1013.340,107.947,-122.582,166.146,58.261,160.590
C02325=1013.344,108.196,-122.598,166.149,58.250,160.589
C02326=1013.348,108.446,-122.615,166.151,58.240,160.587
C02327=1013.352,108.695,-122.631,166.153,58.229,160.585
C02328=1013.356,108.944,-122.648,166.156,58.218,160.584
C02329=1013.361,109.193,-122.665,166.158,58.207,160.582
C02330=1013.364,109.443,-122.681,166.161,58.196,160.581
C02331=1013.369,109.693,-122.698,166.164,58.185,160.579
C02332=1013.374,109.942,-122.715,166.166,58.174,160.578
C02333=1013.377,110.191,-122.732,166.168,58.163,160.576
C02334=1013.381,110.440,-122.749,166.171,58.152,160.575
C02335=1013.385,110.690,-122.766,166.174,58.141,160.573
C02336=1013.390,110.939,-122.782,166.177,58.130,160.572
C02337=1013.394,111.189,-122.799,166.179,58.119,160.570
C02338=1013.398,111.439,-122.816,166.181,58.108,160.569
C02339=1013.402,111.688,-122.833,166.184,58.098,160.567
C02340=1013.406,111.937,-122.850,166.187,58.086,160.566
C02341=1013.410,112.186,-122.867,166.189,58.075,160.564
C02342=1013.415,112.436,-122.885,166.192,58.065,160.563
C02343=1013.419,112.685,-122.902,166.194,58.054,160.561
C02344=1013.422,112.935,-122.919,166.196,58.043,160.560
C02345=1013.426,113.184,-122.936,166.199,58.032,160.558
C02346=1013.430,113.433,-122.953,166.202,58.021,160.557
C02347=1013.435,113.683,-122.970,166.205,58.010,160.555
C02348=1013.439,113.932,-122.988,166.207,57.999,160.554
C02349=1013.443,114.181,-123.005,166.209,57.988,160.552
C02350=1013.447,114.430,-123.022,166.212,57.977,160.551
C02351=1013.451,114.680,-123.040,166.215,57.966,160.549
C02352=1013.455,114.930,-123.057,166.218,57.955,160.548
C02353=1013.459,115.179,-123.074,166.220,57.945,160.546
C02354=1013.463,115.428,-123.091,166.222,57.934,160.545
C02355=1013.467,115.678,-123.108,166.226,57.923,160.543
C02356=1013.471,115.927,-123.125,166.228,57.911,160.541
C02357=1013.475,116.176,-123.143,166.230,57.900,160.540
C02358=1013.479,116.425,-123.160,166.233,57.889,160.538
C02359=1013.484,116.675,-123.178,166.236,57.878,160.537
C02360=1013.487,116.924,-123.195,166.238,57.867,160.536
C02361=1013.491,117.174,-123.212,166.241,57.857,160.534
C02362=1013.495,117.423,-123.229,166.243,57.846,160.532
C02363=1013.500,117.673,-123.246,166.246,57.834,160.531
C02364=1013.504,117.922,-123.264,166.249,57.823,160.529
C02365=1013.508,118.171,-123.281,166.251,57.812,160.528
C02366=1013.511,118.421,-123.299,166.255,57.801,160.526
C02367=1013.515,118.670,-123.316,166.256,57.789,160.525
C02368=1013.519,118.920,-123.334,166.260,57.778,160.523
C02369=1013.523,119.168,-123.351,166.262,57.767,160.522
C02370=1013.528,119.418,-123.369,166.265,57.757,160.520
C02371=1013.532,119.668,-123.386,166.268,57.745,160.519
C02372=1013.536,119.917,-123.403,166.270,57.734,160.517
C02373=1013.540,120.167,-123.420,166.273,57.723,160.516
C02374=1013.544,120.415,-123.438,166.276,57.712,160.514
C02375=1013.548,120.665,-123.455,166.278,57.700,160.512
C02376=1013.553,120.915,-123.473,166.282,57.689,160.511
C02377=1013.556,121.164,-123.490,166.284,57.678,160.510
C02378=1013.561,121.413,-123.508,166.287,57.666,160.508
C02379=1013.565,121.663,-123.525,166.290,57.656,160.506
C02380=1013.569,121.912,-123.542,166.291,57.644,160.505
C02381=1013.574,122.191,-123.561,166.295,57.632,160.503
C02382=1013.578,122.471,-123.581,166.298,57.619,160.501
C02383=1013.584,122.752,-123.600,166.302,57.607,160.500
C02384=1013.588,123.032,-123.620,166.305,57.594,160.498
C02385=1013.592,123.280,-123.638,166.307,57.582,160.496
C02386=1013.597,123.530,-123.655,166.311,57.571,160.495
C02387=1013.600,123.780,-123.673,166.313,57.560,160.493
C02388=1013.605,124.028,-123.690,166.316,57.548,160.492
C02389=1013.609,124.278,-123.708,166.319,57.538,160.490
C02390=1013.613,124.527,-123.725,166.322,57.526,160.489
C02391=1013.617,124.777,-123.742,166.324,57.515,160.487
C02392=1013.622,125.026,-123.760,166.327,57.503,160.485
C02393=1013.626,125.275,-123.777,166.330,57.492,160.484
C02394=1013.630,125.525,-123.795,166.333,57.480,160.482
C02395=1013.634,125.774,-123.812,166.335,57.470,160.481
C02396=1013.639,126.024,-123.830,166.338,57.458,160.479
C02397=1013.643,126.273,-123.848,166.342,57.447,160.478
C02398=1013.647,126.522,-123.865,166.344,57.435,160.476
C02399=1013.651,126.772,-123.882,166.347,57.423,160.474
C02400=1013.655,127.020,-123.900,166.349,57.412,160.473
C02401=1013.660,127.270,-123.917,166.352,57.401,160.471
C02402=1013.664,127.520,-123.934,166.356,57.389,160.470
C02403=1013.668,127.769,-123.953,166.358,57.378,160.468
C02404=1013.672,128.018,-123.970,166.361,57.366,160.467
C02405=1013.677,128.268,-123.988,166.365,57.355,160.465
C02406=1013.681,128.517,-124.005,166.367,57.343,160.464
C02407=1013.685,128.766,-124.022,166.370,57.332,160.462
C02408=1013.690,129.016,-124.040,166.373,57.320,160.461
C02409=1013.694,129.265,-124.057,166.375,57.309,160.459
C02410=1013.698,129.515,-124.076,166.379,57.298,160.458
C02411=1013.702,129.765,-124.093,166.381,57.286,160.456
C02412=1013.705,130.013,-124.112,166.384,57.275,160.454
C02413=1013.710,130.263,-124.130,166.388,57.263,160.453
C02414=1013.714,130.512,-124.147,166.390,57.253,160.451
C02415=1013.718,130.762,-124.166,166.393,57.241,160.450
C02416=1013.722,131.010,-124.184,166.396,57.230,160.448
C02417=1013.727,131.260,-124.201,166.399,57.218,160.447
C02418=1013.730,131.509,-124.219,166.403,57.207,160.445
C02419=1013.735,131.759,-124.238,166.405,57.196,160.444
C02420=1013.738,132.008,-124.255,166.408,57.185,160.442
C02421=1013.743,132.258,-124.273,166.410,57.173,160.440
C02422=1013.747,132.506,-124.291,166.413,57.161,160.439
C02423=1013.751,132.756,-124.310,166.417,57.150,160.438
C02424=1013.755,133.005,-124.327,166.419,57.139,160.436
C02425=1013.760,133.255,-124.345,166.423,57.128,160.435
C02426=1013.763,133.503,-124.364,166.426,57.116,160.433
C02427=1013.768,133.753,-124.381,166.428,57.104,160.431
C02428=1013.771,134.002,-124.400,166.432,57.093,160.430
C02429=1013.776,134.252,-124.418,166.435,57.081,160.428
C02430=1013.780,134.500,-124.435,166.437,57.070,160.427
C02431=1013.784,134.751,-124.454,166.440,57.059,160.425
C02432=1013.789,135.000,-124.472,166.444,57.047,160.424
C02433=1013.792,135.249,-124.490,166.447,57.035,160.422
C02434=1013.797,135.498,-124.508,166.449,57.025,160.421
C02435=1013.800,135.747,-124.527,166.453,57.013,160.419
C02436=1013.805,135.997,-124.544,166.456,57.001,160.417
C02437=1013.809,136.246,-124.562,166.458,56.990,160.416
C02438=1013.813,136.496,-124.581,166.461,56.979,160.414
C02439=1013.818,136.745,-124.599,166.465,56.967,160.413
C02440=1013.821,136.994,-124.617,166.468,56.956,160.411
C02441=1013.826,137.243,-124.635,166.470,56.944,160.410
C02442=1013.829,137.492,-124.654,166.474,56.932,160.408
C02443=1013.834,137.742,-124.671,166.477,56.921,160.407
C02444=1013.838,137.992,-124.690,166.481,56.910,160.405
C02445=1013.843,138.271,-124.711,166.483,56.897,160.403
C02446=1013.847,138.551,-124.732,166.487,56.884,160.402
C02447=1013.851,138.831,-124.752,166.490,56.871,160.400
C02448=1013.857,139.111,-124.773,166.494,56.858,160.398
C02449=1013.861,139.361,-124.792,166.497,56.848,160.397
C02450=1013.864,139.609,-124.810,166.500,56.836,160.395
C02451=1013.869,139.859,-124.828,166.503,56.824,160.394
C02452=1013.872,140.108,-124.847,166.506,56.812,160.392
C02453=1013.876,140.357,-124.865,166.509,56.802,160.391
C02454=1013.881,140.607,-124.884,166.512,56.790,160.389
C02455=1013.885,140.856,-124.902,166.516,56.778,160.388
C02456=1013.889,141.105,-124.920,166.519,56.767,160.386
C02457=1013.893,141.355,-124.939,166.522,56.755,160.385
C02458=1013.897,141.604,-124.957,166.525,56.744,160.383
C02459=1013.902,141.853,-124.975,166.528,56.732,160.381
C02460=1013.906,142.103,-124.994,166.532,56.721,160.380
C02461=1013.909,142.352,-125.013,166.535,56.709,160.379
C02462=1013.914,142.601,-125.031,166.538,56.698,160.377
C02463=1013.918,142.850,-125.050,166.540,56.686,160.375
C02464=1013.922,143.100,-125.069,166.544,56.674,160.374
C02465=1013.926,143.348,-125.087,166.547,56.663,160.372
C02466=1013.930,143.598,-125.106,166.551,56.652,160.371
C02467=1013.934,143.848,-125.124,166.554,56.640,160.369
C02468=1013.939,144.096,-125.142,166.557,56.628,160.368
C02469=1013.943,144.346,-125.161,166.560,56.616,160.366
C02470=1013.947,144.596,-125.180,166.564,56.605,160.365
C02471=1013.952,144.844,-125.198,166.566,56.594,160.363
C02472=1013.955,145.093,-125.217,166.570,56.582,160.362
C02473=1013.959,145.343,-125.236,166.573,56.571,160.360
C02474=1013.963,145.593,-125.254,166.576,56.559,160.358
C02475=1013.968,145.841,-125.273,166.580,56.548,160.357
C02476=1013.972,146.090,-125.292,166.583,56.536,160.356
C02477=1013.976,146.340,-125.310,166.587,56.524,160.354
C02478=1013.980,146.590,-125.329,166.589,56.513,160.352
C02479=1013.984,146.839,-125.349,166.592,56.501,160.351
C02480=1013.988,147.088,-125.367,166.596,56.490,160.350
C02481=1013.992,147.337,-125.386,166.599,56.479,160.348
C02482=1013.997,147.586,-125.405,166.603,56.467,160.346
C02483=1014.001,147.836,-125.423,166.606,56.455,160.345
C02484=1014.005,148.085,-125.442,166.609,56.444,160.343
C02485=1014.009,148.334,-125.461,166.612,56.432,160.342
C02486=1014.013,148.583,-125.480,166.615,56.421,160.340
C02487=1014.017,148.833,-125.499,166.619,56.410,160.339
C02488=1014.021,149.082,-125.518,166.622,56.398,160.337
C02489=1014.025,149.332,-125.537,166.625,56.386,160.336
C02490=1014.029,149.580,-125.556,166.629,56.374,160.334
C02491=1014.033,149.830,-125.575,166.632,56.364,160.333
C02492=1014.037,150.079,-125.594,166.636,56.352,160.331
C02493=1014.041,150.329,-125.613,166.639,56.340,160.330
C02494=1014.046,150.578,-125.633,166.642,56.328,160.328
C02495=1014.050,150.827,-125.651,166.646,56.317,160.327
C02496=1014.054,151.075,-125.670,166.649,56.305,160.325
C02497=1014.058,151.325,-125.689,166.652,56.293,160.324
C02498=1014.063,151.574,-125.708,166.656,56.282,160.322
C02499=1014.067,151.824,-125.727,166.660,56.271,160.321
C02500=1014.071,152.073,-125.746,166.663,56.259,160.319
C02501=1014.075,152.322,-125.765,166.666,56.247,160.318
C02502=1014.079,152.571,-125.785,166.670,56.236,160.316
C02503=1014.083,152.820,-125.803,166.673,56.224,160.315
C02504=1014.087,153.069,-125.822,166.676,56.212,160.313
C02505=1014.091,153.319,-125.841,166.679,56.201,160.311
C02506=1014.095,153.568,-125.861,166.682,56.189,160.310
C02507=1014.099,153.817,-125.881,166.686,56.179,160.309
C02508=1014.103,154.067,-125.899,166.689,56.167,160.307
C02509=1014.108,154.347,-125.922,166.694,56.154,160.306
C02510=1014.113,154.627,-125.943,166.698,56.140,160.304
C02511=1014.118,154.907,-125.964,166.702,56.127,160.302
C02512=1014.122,155.187,-125.986,166.706,56.115,160.301
C02513=1014.126,155.436,-126.005,166.709,56.103,160.299
C02514=1014.131,155.685,-126.025,166.712,56.091,160.297
C02515=1014.134,155.934,-126.043,166.716,56.080,160.296
C02516=1014.139,156.183,-126.063,166.719,56.068,160.294
C02517=1014.143,156.432,-126.082,166.723,56.056,160.293
C02518=1014.146,156.682,-126.101,166.726,56.045,160.291
C02519=1014.151,156.931,-126.121,166.729,56.033,160.290
C02520=1014.155,157.180,-126.140,166.733,56.021,160.288
C02521=1014.159,157.429,-126.160,166.736,56.010,160.287
C02522=1014.163,157.679,-126.179,166.740,55.998,160.285
C02523=1014.168,157.928,-126.198,166.743,55.987,160.284
C02524=1014.172,158.177,-126.218,166.747,55.976,160.282
C02525=1014.176,158.426,-126.238,166.751,55.964,160.281
C02526=1014.180,158.675,-126.257,166.754,55.952,160.279
C02527=1014.184,158.925,-126.277,166.757,55.941,160.278
C02528=1014.187,159.174,-126.297,166.761,55.929,160.276
C02529=1014.192,159.423,-126.317,166.765,55.918,160.275
C02530=1014.195,159.672,-126.337,166.768,55.907,160.274
C02531=1014.200,159.921,-126.356,166.772,55.895,160.272
C02532=1014.203,160.171,-126.376,166.775,55.884,160.271
C02533=1014.208,160.420,-126.396,166.779,55.873,160.269
C02534=1014.211,160.669,-126.416,166.783,55.861,160.268
C02535=1014.215,160.918,-126.436,166.786,55.849,160.266
C02536=1014.219,161.168,-126.455,166.790,55.838,160.265
C02537=1014.223,161.417,-126.475,166.794,55.827,160.264
C02538=1014.227,161.666,-126.495,166.797,55.815,160.262
C02539=1014.231,161.915,-126.515,166.801,55.804,160.261
C02540=1014.235,162.164,-126.534,166.804,55.792,160.259
C02541=1014.240,162.414,-126.556,166.808,55.781,160.257
C02542=1014.243,162.663,-126.576,166.811,55.769,160.256
C02543=1014.247,162.912,-126.595,166.815,55.758,160.255
C02544=1014.251,163.162,-126.615,166.819,55.747,160.253
C02545=1014.255,163.411,-126.635,166.822,55.735,160.252
C02546=1014.259,163.660,-126.655,166.826,55.723,160.250
C02547=1014.264,163.908,-126.675,166.829,55.712,160.249
C02548=1014.267,164.158,-126.695,166.833,55.700,160.247
C02549=1014.271,164.407,-126.715,166.837,55.689,160.246
C02550=1014.275,164.656,-126.735,166.840,55.678,160.244
C02551=1014.279,164.905,-126.755,166.845,55.666,160.243
C02552=1014.283,165.154,-126.774,166.848,55.654,160.242
C02553=1014.287,165.403,-126.795,166.852,55.643,160.240
C02554=1014.292,165.653,-126.815,166.855,55.631,160.239
C02555=1014.296,165.902,-126.835,166.859,55.620,160.237
C02556=1014.299,166.152,-126.855,166.863,55.608,160.236
C02557=1014.304,166.400,-126.875,166.866,55.597,160.234
C02558=1014.308,166.649,-126.895,166.870,55.586,160.233
C02559=1014.312,166.898,-126.915,166.874,55.574,160.231
C02560=1014.316,167.148,-126.935,166.878,55.562,160.230
C02561=1014.319,167.397,-126.955,166.882,55.551,160.228
C02562=1014.324,167.646,-126.975,166.885,55.539,160.227
C02563=1014.328,167.896,-126.995,166.889,55.528,160.225
C02564=1014.333,168.144,-127.016,166.893,55.516,160.224
C02565=1014.336,168.393,-127.036,166.896,55.505,160.222
C02566=1014.341,168.642,-127.055,166.901,55.493,160.221
C02567=1014.345,168.892,-127.076,166.904,55.481,160.220
C02568=1014.349,169.141,-127.096,166.908,55.470,160.218
C02569=1014.353,169.390,-127.116,166.912,55.458,160.217
C02570=1014.357,169.639,-127.137,166.915,55.447,160.215
C02571=1014.361,169.888,-127.156,166.920,55.435,160.214
C02572=1014.366,170.138,-127.176,166.923,55.423,160.212
C02573=1014.370,170.418,-127.199,166.927,55.411,160.211
C02574=1014.375,170.697,-127.222,166.933,55.397,160.209
C02575=1014.379,170.976,-127.245,166.936,55.384,160.207
C02576=1014.384,171.256,-127.267,166.940,55.372,160.206
C02577=1014.388,171.505,-127.287,166.945,55.360,160.204
C02578=1014.393,171.755,-127.308,166.949,55.348,160.203
C02579=1014.397,172.004,-127.328,166.952,55.337,160.201
C02580=1014.401,172.253,-127.348,166.956,55.325,160.200
C02581=1014.405,172.502,-127.368,166.960,55.313,160.199
C02582=1014.409,172.751,-127.389,166.964,55.302,160.197
C02583=1014.414,173.000,-127.408,166.968,55.290,160.196
C02584=1014.417,173.249,-127.429,166.972,55.278,160.194
C02585=1014.422,173.499,-127.450,166.976,55.267,160.193
C02586=1014.426,173.748,-127.469,166.980,55.255,160.191
C02587=1014.430,173.997,-127.490,166.984,55.244,160.190
C02588=1014.435,174.246,-127.510,166.988,55.232,160.188
C02589=1014.439,174.495,-127.531,166.992,55.221,160.187
C02590=1014.443,174.744,-127.550,166.996,55.209,160.186
C02591=1014.447,174.993,-127.571,167.000,55.197,160.184
C02592=1014.452,175.243,-127.591,167.003,55.185,160.182
C02593=1014.456,175.491,-127.611,167.008,55.173,160.181
C02594=1014.461,175.741,-127.633,167.011,55.162,160.180
C02595=1014.465,175.990,-127.652,167.015,55.150,160.178
C02596=1014.469,176.239,-127.673,167.020,55.138,160.177
C02597=1014.473,176.489,-127.693,167.024,55.127,160.175
C02598=1014.478,176.737,-127.713,167.028,55.115,160.174
C02599=1014.481,176.986,-127.734,167.032,55.104,160.173
C02600=1014.487,177.236,-127.754,167.036,55.092,160.171
C02601=1014.491,177.484,-127.775,167.040,55.080,160.170
C02602=1014.495,177.734,-127.795,167.044,55.069,160.168
C02603=1014.499,177.983,-127.815,167.049,55.057,160.167
C02604=1014.503,178.232,-127.836,167.052,55.045,160.165
C02605=1014.508,178.481,-127.856,167.056,55.034,160.164
C02606=1014.512,178.730,-127.877,167.060,55.022,160.162
C02607=1014.516,178.980,-127.897,167.064,55.010,160.161
C02608=1014.521,179.228,-127.918,167.069,54.998,160.160
C02609=1014.526,179.478,-127.939,167.073,54.987,160.158
C02610=1014.530,179.726,-127.959,167.077,54.975,160.157
C02611=1014.534,179.976,-127.979,167.081,54.964,160.155
C02612=1014.538,180.225,-128.000,167.085,54.951,160.154
C02613=1014.543,180.474,-128.020,167.089,54.940,160.152
C02614=1014.547,180.724,-128.041,167.094,54.928,160.151
C02615=1014.552,180.972,-128.061,167.097,54.917,160.149
C02616=1014.556,181.221,-128.082,167.102,54.905,160.148
C02617=1014.560,181.470,-128.103,167.106,54.893,160.147
C02618=1014.565,181.720,-128.123,167.111,54.882,160.145
C02619=1014.569,181.969,-128.144,167.114,54.870,160.144
C02620=1014.573,182.218,-128.166,167.118,54.859,160.142
C02621=1014.577,182.468,-128.188,167.122,54.847,160.141
C02622=1014.581,182.716,-128.208,167.127,54.836,160.140
C02623=1014.585,182.965,-128.229,167.131,54.825,160.138
C02624=1014.589,183.215,-128.251,167.135,54.814,160.137
C02625=1014.593,183.463,-128.272,167.140,54.802,160.135
C02626=1014.597,183.713,-128.293,167.143,54.790,160.134
C02627=1014.601,183.962,-128.314,167.147,54.779,160.133
C02628=1014.605,184.211,-128.336,167.152,54.768,160.131
C02629=1014.609,184.460,-128.357,167.156,54.757,160.130
C02630=1014.614,184.709,-128.378,167.160,54.745,160.129
C02631=1014.618,184.958,-128.399,167.165,54.733,160.127
C02632=1014.621,185.207,-128.421,167.169,54.722,160.126
C02633=1014.626,185.456,-128.442,167.172,54.711,160.124
C02634=1014.630,185.705,-128.463,167.177,54.699,160.123
C02635=1014.635,185.954,-128.484,167.181,54.688,160.122
C02636=1014.638,186.203,-128.506,167.186,54.676,160.120
C02637=1014.643,186.483,-128.530,167.190,54.663,160.119
C02638=1014.647,186.762,-128.554,167.196,54.650,160.117
C02639=1014.652,187.042,-128.578,167.200,54.638,160.116
C02640=1014.657,187.321,-128.602,167.205,54.625,160.114
C02641=1014.661,187.571,-128.623,167.209,54.614,160.113
C02642=1014.665,187.819,-128.644,167.214,54.602,160.111
C02643=1014.669,188.069,-128.666,167.218,54.591,160.110
C02644=1014.674,188.318,-128.687,167.223,54.579,160.109
C02645=1014.678,188.566,-128.709,167.226,54.568,160.107
C02646=1014.682,188.815,-128.730,167.231,54.556,160.106
C02647=1014.686,189.065,-128.751,167.236,54.545,160.105
C02648=1014.690,189.313,-128.773,167.239,54.534,160.103
C02649=1014.695,189.563,-128.794,167.244,54.522,160.102
C02650=1014.698,189.811,-128.816,167.248,54.511,160.100
C02651=1014.703,190.061,-128.837,167.253,54.499,160.099
C02652=1014.707,190.310,-128.859,167.257,54.488,160.098
C02653=1014.712,190.559,-128.880,167.262,54.476,160.096
C02654=1014.715,190.808,-128.902,167.266,54.465,160.095
C02655=1014.720,191.057,-128.924,167.270,54.453,160.093
C02656=1014.725,191.306,-128.945,167.274,54.442,160.092
C02657=1014.729,191.554,-128.966,167.279,54.430,160.091
C02658=1014.733,191.804,-128.988,167.284,54.418,160.089
C02659=1014.737,192.053,-129.009,167.288,54.408,160.088
C02660=1014.741,192.302,-129.031,167.293,54.396,160.087
C02661=1014.745,192.551,-129.052,167.297,54.385,160.085
C02662=1014.750,192.800,-129.074,167.302,54.373,160.084
C02663=1014.755,193.050,-129.095,167.306,54.362,160.083
C02664=1014.759,193.298,-129.117,167.311,54.350,160.081
C02665=1014.763,193.547,-129.139,167.315,54.339,160.080
C02666=1014.767,193.796,-129.161,167.320,54.327,160.079
C02667=1014.772,194.045,-129.182,167.325,54.316,160.077
C02668=1014.776,194.294,-129.203,167.329,54.304,160.076
C02669=1014.780,194.543,-129.226,167.334,54.293,160.074
C02670=1014.785,194.792,-129.247,167.337,54.281,160.073
C02671=1014.790,195.041,-129.269,167.342,54.270,160.072
C02672=1014.793,195.291,-129.290,167.347,54.258,160.070
C02673=1014.798,195.540,-129.312,167.351,54.247,160.069
C02674=1014.802,195.788,-129.334,167.356,54.235,160.068
C02675=1014.807,196.037,-129.355,167.362,54.224,160.067
C02676=1014.811,196.286,-129.377,167.365,54.213,160.065
C02677=1014.816,196.535,-129.399,167.370,54.201,160.064
C02678=1014.820,196.785,-129.420,167.375,54.190,160.062
C02679=1014.824,197.034,-129.443,167.379,54.178,160.061
C02680=1014.829,197.282,-129.464,167.384,54.167,160.060
C02681=1014.833,197.531,-129.485,167.389,54.155,160.058
C02682=1014.838,197.780,-129.507,167.393,54.144,160.057
C02683=1014.842,198.029,-129.530,167.398,54.132,160.056
C02684=1014.847,198.279,-129.551,167.403,54.121,160.054
C02685=1014.851,198.528,-129.573,167.407,54.109,160.053
C02686=1014.856,198.777,-129.595,167.412,54.098,160.052
C02687=1014.860,199.025,-129.617,167.417,54.086,160.050
C02688=1014.864,199.275,-129.639,167.421,54.075,160.049
C02689=1014.869,199.524,-129.661,167.426,54.063,160.047
C02690=1014.872,199.772,-129.683,167.431,54.052,160.046
C02691=1014.877,200.022,-129.705,167.435,54.041,160.045
C02692=1014.881,200.270,-129.727,167.440,54.029,160.044
C02693=1014.885,200.520,-129.750,167.444,54.018,160.042
C02694=1014.890,200.769,-129.772,167.449,54.007,160.041
C02695=1014.894,201.017,-129.794,167.455,53.996,160.040
C02696=1014.898,201.267,-129.816,167.459,53.985,160.038
C02697=1014.903,201.516,-129.839,167.464,53.973,160.037
C02698=1014.907,201.765,-129.861,167.469,53.961,160.036
C02699=1014.911,202.014,-129.883,167.473,53.951,160.035
C02700=1014.916,202.262,-129.906,167.478,53.939,160.033
C02701=1014.935,203.369,-130.005,167.998,54.006,160.161
C02702=1014.941,203.601,-130.027,168.002,53.997,160.160
C02703=1014.945,203.833,-130.049,168.006,53.987,160.159
C02704=1014.950,204.064,-130.072,168.010,53.978,160.158
C02705=1014.956,204.297,-130.094,168.014,53.968,160.157
C02706=1014.960,204.529,-130.117,168.018,53.959,160.155
C02707=1014.966,204.760,-130.139,168.022,53.949,160.154
C02708=1014.971,204.993,-130.161,168.026,53.940,160.153
C02709=1014.976,205.225,-130.184,168.031,53.930,160.152
C02710=1014.981,205.473,-130.208,168.034,53.920,160.151
C02711=1014.986,205.722,-130.232,168.039,53.910,160.149
C02712=1014.992,205.972,-130.256,168.043,53.900,160.148
C02713=1014.997,206.220,-130.280,168.048,53.890,160.147
C02714=1015.002,206.469,-130.305,168.053,53.880,160.146
C02715=1015.008,206.717,-130.329,168.056,53.870,160.145
C02716=1015.013,206.966,-130.353,168.060,53.859,160.143
C02717=1015.018,207.215,-130.377,168.065,53.850,160.142
C02718=1015.024,207.463,-130.402,168.070,53.839,160.141
C02719=1015.030,207.712,-130.426,168.074,53.830,160.140
C02720=1015.035,207.961,-130.450,168.078,53.819,160.138
C02721=1015.040,208.210,-130.475,168.083,53.810,160.137
C02722=1015.045,208.458,-130.499,168.086,53.800,160.136
C02723=1015.051,208.707,-130.523,168.091,53.790,160.135
C02724=1015.057,208.956,-130.548,168.096,53.780,160.134
C02725=1015.062,209.205,-130.572,168.100,53.770,160.133
C02726=1015.067,209.453,-130.596,168.104,53.760,160.131
C02727=1015.073,209.702,-130.621,168.109,53.751,160.130
C02728=1015.078,209.951,-130.646,168.113,53.741,160.129
C02729=1015.083,210.200,-130.670,168.117,53.731,160.128
C02730=1015.088,210.449,-130.694,168.122,53.721,160.127
C02731=1015.094,210.697,-130.719,168.126,53.711,160.125
C02732=1015.099,210.946,-130.743,168.131,53.701,160.124
C02733=1015.104,211.195,-130.769,168.135,53.692,160.123
C02734=1015.110,211.443,-130.793,168.139,53.682,160.122
C02735=1015.115,211.692,-130.817,168.143,53.673,160.121
C02736=1015.121,211.941,-130.842,168.148,53.663,160.120
C02737=1015.125,212.190,-130.867,168.153,53.653,160.119
C02738=1015.131,212.438,-130.892,168.157,53.644,160.117
C02739=1015.136,212.687,-130.916,168.162,53.634,160.116
C02740=1015.142,212.936,-130.941,168.165,53.625,160.115
C02741=1015.147,213.185,-130.966,168.170,53.615,160.114
C02742=1015.152,213.433,-130.990,168.174,53.606,160.113
C02743=1015.158,213.682,-131.015,168.179,53.596,160.112
C02744=1015.164,213.931,-131.039,168.183,53.587,160.111
C02745=1015.169,214.179,-131.064,168.188,53.576,160.109
C02746=1015.174,214.428,-131.090,168.191,53.567,160.108
C02747=1015.180,214.677,-131.114,168.196,53.557,160.107
C02748=1015.186,214.926,-131.138,168.200,53.548,160.106
C02749=1015.191,215.174,-131.163,168.205,53.538,160.105
C02750=1015.196,215.423,-131.188,168.209,53.529,160.104
C02751=1015.202,215.672,-131.213,168.214,53.519,160.103
C02752=1015.207,215.920,-131.238,168.218,53.510,160.102
C02753=1015.213,216.169,-131.262,168.223,53.500,160.101
C02754=1015.218,216.418,-131.287,168.227,53.491,160.099
C02755=1015.223,216.666,-131.312,168.232,53.482,160.099
C02756=1015.229,216.916,-131.337,168.236,53.473,160.097
C02757=1015.235,217.164,-131.362,168.241,53.463,160.096
C02758=1015.240,217.413,-131.387,168.245,53.454,160.095
C02759=1015.246,217.661,-131.412,168.250,53.444,160.094
C02760=1015.251,217.910,-131.436,168.254,53.435,160.093
C02761=1015.256,218.159,-131.462,168.258,53.426,160.092
C02762=1015.262,218.402,-131.486,168.263,53.417,160.091
C02763=1015.267,218.646,-131.511,168.267,53.407,160.090
C02764=1015.272,218.889,-131.536,168.272,53.399,160.089
C02765=1015.278,219.133,-131.560,168.276,53.390,160.088
C02766=1015.283,219.377,-131.585,168.280,53.381,160.087
C02767=1015.288,219.620,-131.610,168.284,53.372,160.086
C02768=1015.293,219.864,-131.635,168.289,53.363,160.085
C02769=1015.298,220.107,-131.659,168.294,53.353,160.084
C02770=1015.304,220.356,-131.685,168.298,53.345,160.083
C02771=1015.309,220.605,-131.709,168.302,53.336,160.082
C02772=1015.315,220.854,-131.735,168.306,53.327,160.081
C02773=1015.320,221.102,-131.760,168.311,53.317,160.080
C02774=1015.326,221.351,-131.786,168.316,53.309,160.079
C02775=1015.331,221.599,-131.810,168.320,53.300,160.077
C02776=1015.336,221.848,-131.836,168.325,53.290,160.076
C02777=1015.342,222.097,-131.862,168.329,53.281,160.076
C02778=1015.348,222.345,-131.887,168.333,53.272,160.074
C02779=1015.353,222.595,-131.912,168.338,53.264,160.073
C02780=1015.358,222.843,-131.937,168.343,53.254,160.072
C02781=1015.364,223.092,-131.963,168.347,53.245,160.071
C02782=1015.369,223.340,-131.988,168.351,53.237,160.071
C02783=1015.375,223.589,-132.014,168.355,53.228,160.069
C02784=1015.381,223.838,-132.039,168.361,53.219,160.069
C02785=1015.386,224.086,-132.064,168.365,53.210,160.067
C02786=1015.392,224.335,-132.089,168.369,53.201,160.066
C02787=1015.397,224.583,-132.115,168.373,53.192,160.065
C02788=1015.402,224.832,-132.141,168.379,53.183,160.064
C02789=1015.408,225.081,-132.166,168.383,53.174,160.064
C02790=1015.413,225.329,-132.192,168.387,53.165,160.062
C02791=1015.419,225.578,-132.216,168.392,53.157,160.061
C02792=1015.425,225.827,-132.242,168.396,53.148,160.060
C02793=1015.430,226.075,-132.267,168.401,53.138,160.059
C02794=1015.436,226.324,-132.293,168.406,53.130,160.058
C02795=1015.441,226.573,-132.319,168.410,53.121,160.058
C02796=1015.446,226.822,-132.345,168.415,53.113,160.057
C02797=1015.453,227.070,-132.371,168.419,53.104,160.056
C02798=1015.457,227.318,-132.396,168.423,53.095,160.055
C02799=1015.463,227.567,-132.422,168.428,53.087,160.054
C02800=1015.468,227.816,-132.448,168.433,53.078,160.053
C02801=1015.474,228.065,-132.474,168.438,53.069,160.052
C02802=1015.479,228.313,-132.499,168.442,53.061,160.051
C02803=1015.485,228.562,-132.525,168.446,53.052,160.050
C02804=1015.490,228.811,-132.551,168.451,53.044,160.049
C02805=1015.496,229.058,-132.577,168.455,53.035,160.048
C02806=1015.501,229.307,-132.603,168.460,53.027,160.047
C02807=1015.507,229.556,-132.629,168.464,53.018,160.046
C02808=1015.512,229.804,-132.654,168.469,53.010,160.045
C02809=1015.518,230.053,-132.681,168.473,53.001,160.044
C02810=1015.523,230.302,-132.707,168.478,52.993,160.043
C02811=1015.529,230.551,-132.733,168.482,52.984,160.043
C02812=1015.534,230.799,-132.758,168.487,52.976,160.042
C02813=1015.539,231.047,-132.785,168.491,52.967,160.041
C02814=1015.545,231.296,-132.811,168.496,52.959,160.040
C02815=1015.550,231.545,-132.837,168.500,52.950,160.039
C02816=1015.556,231.793,-132.863,168.505,52.942,160.038
C02817=1015.561,232.042,-132.889,168.510,52.934,160.037
C02818=1015.567,232.290,-132.916,168.514,52.925,160.036
C02819=1015.572,232.539,-132.942,168.519,52.917,160.035
C02820=1015.578,232.788,-132.968,168.523,52.908,160.034
C02821=1015.583,233.036,-132.994,168.528,52.900,160.033
C02822=1015.589,233.275,-133.018,168.533,52.892,160.033
C02823=1015.594,233.515,-133.044,168.537,52.884,160.032
C02824=1015.599,233.755,-133.069,168.541,52.876,160.031
C02825=1015.605,233.994,-133.094,168.546,52.868,160.030
C02826=1015.610,234.234,-133.120,168.551,52.860,160.029
C02827=1015.615,234.474,-133.145,168.554,52.852,160.028
C02828=1015.621,234.712,-133.170,168.559,52.844,160.028
C02829=1015.626,234.952,-133.195,168.564,52.836,160.027
C02830=1015.631,235.200,-133.222,168.569,52.828,160.026
C02831=1015.637,235.449,-133.248,168.572,52.820,160.025
C02832=1015.643,235.697,-133.274,168.577,52.812,160.024
C02833=1015.648,235.946,-133.300,168.582,52.803,160.023
C02834=1015.654,236.195,-133.327,168.586,52.795,160.022
C02835=1015.660,236.443,-133.354,168.591,52.787,160.022
C02836=1015.665,236.692,-133.379,168.596,52.779,160.021
C02837=1015.671,236.940,-133.406,168.601,52.771,160.020
C02838=1015.676,237.189,-133.432,168.605,52.762,160.019
C02839=1015.682,237.437,-133.458,168.610,52.754,160.018
C02840=1015.687,237.685,-133.485,168.615,52.746,160.017
C02841=1015.693,237.934,-133.511,168.619,52.738,160.016
C02842=1015.699,238.183,-133.538,168.623,52.730,160.016
C02843=1015.704,238.431,-133.564,168.628,52.722,160.015
C02844=1015.710,238.679,-133.591,168.633,52.714,160.014
C02845=1015.716,238.928,-133.617,168.638,52.706,160.013
C02846=1015.721,239.177,-133.644,168.642,52.698,160.012
C02847=1015.726,239.425,-133.671,168.647,52.690,160.012
C02848=1015.732,239.674,-133.697,168.651,52.682,160.011
C02849=1015.737,239.923,-133.725,168.656,52.674,160.010
C02850=1015.743,240.171,-133.751,168.661,52.667,160.009
C02851=1015.749,240.419,-133.778,168.666,52.659,160.008
C02852=1015.755,240.668,-133.805,168.670,52.650,160.008
C02853=1015.759,240.917,-133.831,168.674,52.643,160.007
C02854=1015.765,241.165,-133.858,168.679,52.635,160.006
C02855=1015.771,241.414,-133.884,168.684,52.628,160.005
C02856=1015.776,241.662,-133.912,168.689,52.619,160.004
C02857=1015.782,241.911,-133.938,168.693,52.612,160.004
C02858=1015.787,242.159,-133.965,168.698,52.604,160.003
C02859=1015.792,242.408,-133.992,168.703,52.596,160.002
C02860=1015.798,242.656,-134.019,168.708,52.589,160.001
C02861=1015.804,242.904,-134.046,168.711,52.580,160.000
C02862=1015.809,243.152,-134.073,168.716,52.573,160.000
C02863=1015.815,243.401,-134.100,168.721,52.565,159.999
C02864=1015.820,243.649,-134.127,168.726,52.557,159.998
C02865=1015.825,243.898,-134.155,168.730,52.550,159.997
C02866=1015.831,244.146,-134.181,168.735,52.542,159.997
C02867=1015.836,244.395,-134.209,168.740,52.534,159.996
C02868=1015.842,244.643,-134.236,168.744,52.527,159.995
C02869=1015.848,244.892,-134.263,168.749,52.519,159.995
C02870=1015.853,245.141,-134.291,168.754,52.513,159.994
C02871=1015.859,245.389,-134.318,168.759,52.505,159.993
C02872=1015.864,245.637,-134.345,168.764,52.497,159.993
C02873=1015.870,245.886,-134.372,168.768,52.490,159.992
C02874=1015.875,246.134,-134.399,168.773,52.482,159.991
C02875=1015.880,246.382,-134.427,168.778,52.474,159.990
C02876=1015.886,246.632,-134.454,168.782,52.467,159.989
C02877=1015.891,246.880,-134.481,168.787,52.459,159.989
C02878=1015.897,247.128,-134.509,168.792,52.452,159.988
C02879=1015.903,247.377,-134.536,168.796,52.445,159.987
C02880=1015.908,247.625,-134.563,168.801,52.437,159.987
C02881=1015.914,247.873,-134.591,168.806,52.430,159.986
C02882=1015.920,248.149,-134.621,168.811,52.421,159.985
C02883=1015.926,248.424,-134.651,168.816,52.413,159.984
C02884=1015.933,248.700,-134.681,168.822,52.405,159.984
C02885=1015.938,248.975,-134.712,168.827,52.397,159.983
C02886=1015.945,249.223,-134.740,168.832,52.389,159.982
C02887=1015.950,249.472,-134.767,168.837,52.382,159.982
C02888=1015.955,249.720,-134.795,168.841,52.375,159.981
C02889=1015.961,249.969,-134.822,168.846,52.367,159.980
C02890=1015.967,250.217,-134.850,168.850,52.360,159.979
C02891=1015.972,250.465,-134.876,168.856,52.353,159.979
C02892=1015.978,250.713,-134.904,168.861,52.345,159.978
C02893=1015.983,250.963,-134.932,168.865,52.338,159.977
C02894=1015.988,251.184,-134.957,168.869,52.331,159.977
C02895=1015.994,251.408,-134.981,168.874,52.325,159.976
C02896=1015.999,251.630,-135.006,168.879,52.319,159.976
C02897=1016.004,251.853,-135.030,168.882,52.312,159.975
C02898=1016.009,252.075,-135.055,168.887,52.306,159.974
C02899=1016.014,252.298,-135.080,168.891,52.299,159.974
C02900=1016.019,252.520,-135.104,168.896,52.292,159.973
C02901=1016.024,252.743,-135.129,168.900,52.286,159.973
C02902=1016.030,252.991,-135.157,168.904,52.279,159.972
C02903=1016.036,253.240,-135.184,168.910,52.271,159.971
C02904=1016.041,253.488,-135.212,168.914,52.264,159.970
C02905=1016.047,253.737,-135.240,168.919,52.257,159.970
C02906=1016.053,253.985,-135.267,168.924,52.249,159.969
C02907=1016.058,254.234,-135.294,168.929,52.243,159.969
C02908=1016.065,254.482,-135.322,168.934,52.235,159.968
C02909=1016.070,254.730,-135.350,168.938,52.229,159.967
C02910=1016.076,254.979,-135.378,168.944,52.222,159.967
C02911=1016.082,255.227,-135.405,168.948,52.214,159.966
C02912=1016.088,255.475,-135.433,168.953,52.207,159.966
C02913=1016.093,255.724,-135.461,168.958,52.200,159.965
C02914=1016.099,255.972,-135.488,168.963,52.193,159.964
C02915=1016.105,256.221,-135.516,168.968,52.185,159.963
C02916=1016.111,256.469,-135.544,168.972,52.179,159.963
C02917=1016.117,256.718,-135.572,168.978,52.172,159.962
C02918=1016.123,256.966,-135.600,168.982,52.164,159.962
C02919=1016.129,257.215,-135.627,168.987,52.157,159.961
C02920=1016.134,257.463,-135.655,168.993,52.150,159.961
C02921=1016.140,257.711,-135.683,168.997,52.143,159.960
C02922=1016.146,257.959,-135.711,169.002,52.136,159.959
C02923=1016.152,258.208,-135.739,169.007,52.130,159.959
C02924=1016.158,258.456,-135.766,169.012,52.123,159.958
C02925=1016.164,258.704,-135.795,169.016,52.115,159.957
C02926=1016.170,258.952,-135.823,169.022,52.108,159.957
C02927=1016.176,259.201,-135.850,169.026,52.102,159.956
C02928=1016.182,259.449,-135.878,169.032,52.095,159.956
C02929=1016.188,259.697,-135.906,169.036,52.087,159.955
C02930=1016.194,259.945,-135.934,169.041,52.080,159.954
C02931=1016.199,260.195,-135.963,169.046,52.074,159.954
C02932=1016.204,260.443,-135.991,169.051,52.067,159.953
C02933=1016.210,260.691,-136.019,169.056,52.060,159.953
C02934=1016.216,260.939,-136.048,169.060,52.054,159.952
C02935=1016.222,261.188,-136.076,169.066,52.047,159.952
C02936=1016.228,261.436,-136.105,169.070,52.040,159.951
C02937=1016.233,261.684,-136.133,169.076,52.033,159.951
C02938=1016.239,261.932,-136.162,169.080,52.027,159.950
C02939=1016.245,262.180,-136.190,169.086,52.020,159.950
C02940=1016.251,262.429,-136.218,169.091,52.014,159.949
C02941=1016.256,262.678,-136.246,169.095,52.007,159.948
C02942=1016.262,262.912,-136.273,169.100,52.001,159.948
C02943=1016.268,263.148,-136.300,169.105,51.995,159.947
C02944=1016.273,263.383,-136.328,169.109,51.988,159.947
C02945=1016.278,263.618,-136.354,169.114,51.981,159.946
C02946=1016.284,263.853,-136.381,169.119,51.976,159.946
C02947=1016.290,264.088,-136.408,169.123,51.969,159.945
C02948=1016.294,264.324,-136.435,169.128,51.963,159.945
C02949=1016.300,264.559,-136.462,169.133,51.956,159.944
C02950=1016.306,264.807,-136.491,169.139,51.950,159.944
C02951=1016.312,265.055,-136.519,169.143,51.944,159.943
C02952=1016.318,265.304,-136.548,169.149,51.937,159.943
C02953=1016.324,265.552,-136.577,169.153,51.930,159.942
C02954=1016.329,265.800,-136.605,169.158,51.924,159.942
C02955=1016.335,266.048,-136.634,169.164,51.917,159.941
C02956=1016.341,266.297,-136.663,169.168,51.911,159.941
C02957=1016.347,266.545,-136.692,169.173,51.905,159.940
C02958=1016.353,266.792,-136.720,169.179,51.898,159.940
C02959=1016.358,267.042,-136.749,169.184,51.892,159.940
C02960=1016.364,267.290,-136.778,169.188,51.885,159.939
C02961=1016.370,267.538,-136.807,169.194,51.878,159.938
C02962=1016.376,267.786,-136.835,169.199,51.873,159.938
C02963=1016.382,268.034,-136.864,169.204,51.866,159.938
C02964=1016.387,268.283,-136.893,169.209,51.860,159.937
C02965=1016.393,268.531,-136.922,169.214,51.853,159.937
C02966=1016.399,268.779,-136.951,169.220,51.847,159.936
C02967=1016.405,269.027,-136.980,169.224,51.840,159.936
C02968=1016.411,269.276,-137.009,169.229,51.834,159.935
C02969=1016.417,269.524,-137.038,169.234,51.828,159.935
C02970=1016.423,269.772,-137.067,169.240,51.822,159.934
C02971=1016.428,270.020,-137.096,169.244,51.815,159.934
C02972=1016.434,270.268,-137.125,169.249,51.809,159.933
C02973=1016.440,270.516,-137.155,169.255,51.803,159.933
C02974=1016.446,270.765,-137.183,169.259,51.796,159.933
C02975=1016.452,271.013,-137.212,169.264,51.790,159.932
C02976=1016.457,271.262,-137.242,169.270,51.784,159.932
C02977=1016.464,271.510,-137.271,169.275,51.778,159.931
C02978=1016.469,271.758,-137.300,169.280,51.772,159.931
C02979=1016.475,272.006,-137.329,169.285,51.766,159.930
C02980=1016.481,272.254,-137.358,169.290,51.759,159.930
C02981=1016.487,272.502,-137.388,169.295,51.753,159.930
C02982=1016.493,272.750,-137.417,169.300,51.747,159.929
C02983=1016.498,272.999,-137.447,169.305,51.741,159.929
C02984=1016.505,273.247,-137.476,169.311,51.734,159.928
C02985=1016.510,273.495,-137.505,169.316,51.729,159.928
C02986=1016.516,273.744,-137.534,169.321,51.723,159.927
C02987=1016.522,273.992,-137.564,169.327,51.717,159.927
C02988=1016.528,274.240,-137.593,169.332,51.711,159.927
C02989=1016.534,274.489,-137.623,169.337,51.705,159.926
C02990=1016.540,274.736,-137.652,169.341,51.698,159.926
C02991=1016.546,274.985,-137.682,169.347,51.692,159.926
C02992=1016.552,275.233,-137.711,169.352,51.686,159.925
C02993=1016.557,275.481,-137.741,169.357,51.680,159.925
C02994=1016.563,275.729,-137.769,169.362,51.674,159.924
C02995=1016.570,275.976,-137.799,169.368,51.668,159.924
C02996=1016.575,276.225,-137.829,169.373,51.662,159.924
C02997=1016.581,276.473,-137.858,169.378,51.656,159.923
C02998=1016.587,276.721,-137.887,169.383,51.651,159.923
C02999=1016.593,276.969,-137.918,169.389,51.644,159.923
C03000=1016.598,277.217,-137.947,169.394,51.639,159.922
C03001=1016.604,277.465,-137.978,169.399,51.633,159.922
C03002=1016.610,277.703,-138.006,169.404,51.627,159.922
C03003=1016.616,277.940,-138.034,169.409,51.622,159.921
C03004=1016.621,278.178,-138.063,169.414,51.616,159.921
C03005=1016.627,278.416,-138.092,169.418,51.611,159.921
C03006=1016.633,278.652,-138.119,169.423,51.605,159.920
C03007=1016.638,278.890,-138.149,169.429,51.600,159.920
C03008=1016.644,279.127,-138.177,169.434,51.594,159.920
C03009=1016.649,279.365,-138.206,169.439,51.588,159.919
C03010=1016.656,279.612,-138.236,169.444,51.583,159.919
C03011=1016.662,279.861,-138.265,169.449,51.577,159.919
C03012=1016.667,280.109,-138.296,169.455,51.571,159.918
C03013=1016.673,280.357,-138.325,169.460,51.565,159.918
C03014=1016.679,280.605,-138.355,169.465,51.560,159.918
C03015=1016.686,280.854,-138.385,169.470,51.554,159.917
C03016=1016.691,281.102,-138.415,169.475,51.548,159.917
C03017=1016.697,281.349,-138.446,169.481,51.542,159.917
C03018=1016.703,281.598,-138.475,169.487,51.537,159.916
C03019=1016.709,281.845,-138.505,169.492,51.531,159.916
C03020=1016.716,282.094,-138.536,169.497,51.525,159.916
C03021=1016.722,282.342,-138.565,169.502,51.520,159.915
C03022=1016.728,282.590,-138.595,169.508,51.514,159.915
C03023=1016.734,282.838,-138.626,169.513,51.509,159.915
C03024=1016.739,283.086,-138.655,169.518,51.503,159.915
C03025=1016.746,283.334,-138.685,169.523,51.497,159.914
C03026=1016.752,283.582,-138.716,169.529,51.492,159.914
C03027=1016.758,283.830,-138.746,169.535,51.486,159.914
C03028=1016.764,284.079,-138.776,169.540,51.480,159.914
C03029=1016.770,284.327,-138.806,169.545,51.475,159.913
C03030=1016.776,284.575,-138.836,169.551,51.469,159.913
C03031=1016.782,284.822,-138.866,169.556,51.464,159.913
C03032=1016.789,285.071,-138.897,169.561,51.458,159.912
C03033=1016.794,285.319,-138.928,169.567,51.452,159.912
C03034=1016.800,285.567,-138.958,169.572,51.447,159.912
C03035=1016.807,285.815,-138.989,169.578,51.442,159.912
C03036=1016.812,286.063,-139.019,169.583,51.436,159.911
C03037=1016.818,286.311,-139.049,169.588,51.431,159.911
C03038=1016.825,286.559,-139.080,169.594,51.426,159.911
C03039=1016.830,286.807,-139.110,169.600,51.420,159.911
C03040=1016.836,287.055,-139.141,169.605,51.414,159.910
C03041=1016.843,287.303,-139.171,169.610,51.409,159.910
C03042=1016.849,287.551,-139.202,169.615,51.404,159.910
C03043=1016.854,287.799,-139.232,169.621,51.398,159.910
C03044=1016.861,288.048,-139.263,169.626,51.393,159.909
C03045=1016.867,288.295,-139.293,169.632,51.388,159.909
C03046=1016.873,288.543,-139.324,169.638,51.383,159.909
C03047=1016.879,288.791,-139.355,169.643,51.377,159.909
C03048=1016.885,289.039,-139.385,169.648,51.372,159.909
C03049=1016.891,289.287,-139.416,169.654,51.366,159.908
C03050=1016.897,289.535,-139.446,169.659,51.361,159.908
C03051=1016.904,289.783,-139.478,169.665,51.356,159.908
C03052=1016.910,290.031,-139.508,169.670,51.351,159.908
C03053=1016.915,290.280,-139.539,169.675,51.345,159.907
C03054=1016.921,290.528,-139.570,169.681,51.340,159.907
C03055=1016.927,290.775,-139.601,169.687,51.335,159.907
C03056=1016.934,291.023,-139.632,169.692,51.329,159.907
C03057=1016.940,291.271,-139.662,169.698,51.324,159.907
C03058=1016.946,291.519,-139.693,169.703,51.319,159.907
C03059=1016.952,291.767,-139.724,169.708,51.314,159.906
C03060=1016.959,292.015,-139.755,169.714,51.309,159.906
C03061=1016.964,292.263,-139.786,169.719,51.304,159.906
C03062=1016.970,292.506,-139.816,169.725,51.299,159.906
C03063=1016.977,292.750,-139.848,169.730,51.294,159.906
C03064=1016.983,292.993,-139.878,169.736,51.289,159.906
C03065=1016.989,293.237,-139.909,169.741,51.284,159.905
C03066=1016.994,293.480,-139.939,169.747,51.279,159.905
C03067=1017.000,293.724,-139.970,169.752,51.274,159.905
C03068=1017.006,293.967,-140.001,169.758,51.269,159.905
C03069=1017.011,294.211,-140.032,169.763,51.264,159.905
C03070=1017.018,294.459,-140.063,169.769,51.259,159.905
C03071=1017.024,294.706,-140.095,169.774,51.254,159.905
C03072=1017.030,294.955,-140.126,169.780,51.249,159.905
C03073=1017.036,295.203,-140.158,169.786,51.245,159.905
C03074=1017.042,295.450,-140.189,169.791,51.240,159.904
C03075=1017.048,295.698,-140.221,169.797,51.234,159.904
C03076=1017.053,295.946,-140.252,169.802,51.230,159.904
C03077=1017.060,296.194,-140.283,169.808,51.225,159.904
C03078=1017.066,296.443,-140.315,169.814,51.220,159.904
C03079=1017.072,296.690,-140.346,169.819,51.215,159.904
C03080=1017.078,296.938,-140.378,169.825,51.210,159.904
C03081=1017.085,297.186,-140.410,169.831,51.205,159.904
C03082=1017.090,297.434,-140.441,169.837,51.200,159.904
C03083=1017.097,297.681,-140.473,169.842,51.196,159.904
C03084=1017.103,297.930,-140.505,169.848,51.191,159.903
C03085=1017.109,298.177,-140.536,169.854,51.186,159.903
C03086=1017.115,298.425,-140.568,169.859,51.181,159.903
C03087=1017.121,298.673,-140.600,169.865,51.177,159.903
C03088=1017.127,298.920,-140.631,169.870,51.171,159.903
C03089=1017.133,299.169,-140.663,169.876,51.167,159.903
C03090=1017.140,299.417,-140.694,169.882,51.162,159.903
C03091=1017.146,299.665,-140.726,169.887,51.157,159.903
C03092=1017.152,299.913,-140.758,169.893,51.153,159.903
C03093=1017.158,300.160,-140.789,169.899,51.148,159.903
C03094=1017.165,300.408,-140.821,169.904,51.143,159.903
C03095=1017.171,300.656,-140.853,169.910,51.138,159.903
C03096=1017.178,300.904,-140.885,169.917,51.133,159.903
C03097=1017.184,301.152,-140.917,169.923,51.129,159.903
C03098=1017.189,301.399,-140.949,169.928,51.124,159.902
C03099=1017.196,301.647,-140.980,169.934,51.119,159.902
C03100=1017.202,301.895,-141.012,169.940,51.115,159.903
C03101=1017.209,302.143,-141.044,169.945,51.110,159.902
C03102=1017.215,302.391,-141.076,169.951,51.105,159.902
C03103=1017.221,302.639,-141.108,169.957,51.101,159.902
C03104=1017.227,302.887,-141.140,169.962,51.096,159.902
C03105=1017.234,303.134,-141.172,169.968,51.091,159.902
C03106=1017.240,303.382,-141.204,169.974,51.087,159.902
C03107=1017.246,303.630,-141.236,169.981,51.082,159.902
C03108=1017.253,303.877,-141.268,169.986,51.078,159.902
C03109=1017.259,304.126,-141.300,169.992,51.073,159.902
C03110=1017.266,304.373,-141.331,169.998,51.069,159.902
C03111=1017.272,304.621,-141.364,170.003,51.064,159.902
C03112=1017.279,304.869,-141.395,170.009,51.059,159.902
C03113=1017.285,305.117,-141.428,170.015,51.055,159.902
C03114=1017.292,305.364,-141.460,170.021,51.050,159.902
C03115=1017.298,305.613,-141.492,170.027,51.046,159.902
C03116=1017.304,305.860,-141.524,170.033,51.041,159.902
C03117=1017.311,306.108,-141.556,170.039,51.037,159.902
C03118=1017.317,306.356,-141.589,170.045,51.032,159.902
C03119=1017.324,306.604,-141.620,170.051,51.028,159.902
C03120=1017.330,306.851,-141.653,170.057,51.023,159.902
C03121=1017.337,307.100,-141.685,170.063,51.019,159.902
C03122=1017.344,307.357,-141.718,170.068,51.014,159.902
C03123=1017.351,307.613,-141.752,170.075,51.010,159.902
C03124=1017.357,307.870,-141.785,170.081,51.005,159.902
C03125=1017.364,308.127,-141.819,170.088,51.000,159.902
C03126=1017.370,308.375,-141.851,170.094,50.996,159.903
C03127=1017.378,308.623,-141.883,170.100,50.992,159.903
C03128=1017.384,308.870,-141.916,170.105,50.987,159.903
C03129=1017.390,309.119,-141.948,170.111,50.983,159.903
C03130=1017.397,309.366,-141.980,170.117,50.978,159.903
C03131=1017.403,309.613,-142.013,170.123,50.974,159.903
C03132=1017.410,309.861,-142.046,170.129,50.970,159.903
C03133=1017.416,310.109,-142.078,170.135,50.966,159.903
C03134=1017.422,310.356,-142.111,170.141,50.961,159.903
C03135=1017.429,310.604,-142.144,170.147,50.957,159.903
C03136=1017.435,310.852,-142.178,170.153,50.953,159.903
C03137=1017.441,311.100,-142.210,170.159,50.949,159.903
C03138=1017.447,311.348,-142.243,170.165,50.945,159.903
C03139=1017.454,311.595,-142.276,170.171,50.941,159.903
C03140=1017.460,311.842,-142.309,170.177,50.937,159.903
C03141=1017.466,312.091,-142.343,170.183,50.933,159.904
C03142=1017.473,312.338,-142.376,170.189,50.928,159.904
C03143=1017.479,312.586,-142.408,170.196,50.924,159.904
C03144=1017.486,312.833,-142.442,170.202,50.920,159.904
C03145=1017.491,313.081,-142.475,170.208,50.916,159.904
C03146=1017.498,313.329,-142.508,170.214,50.912,159.904
C03147=1017.504,313.577,-142.541,170.220,50.908,159.904
C03148=1017.511,313.824,-142.575,170.227,50.904,159.905
C03149=1017.518,314.072,-142.608,170.232,50.900,159.905
C03150=1017.523,314.320,-142.641,170.239,50.896,159.905
C03151=1017.530,314.567,-142.674,170.245,50.891,159.905
C03152=1017.536,314.814,-142.707,170.251,50.888,159.905
C03153=1017.543,315.063,-142.740,170.257,50.884,159.905
C03154=1017.550,315.310,-142.774,170.263,50.880,159.905
C03155=1017.555,315.558,-142.807,170.269,50.876,159.905
C03156=1017.562,315.805,-142.841,170.275,50.872,159.906
C03157=1017.569,316.053,-142.874,170.282,50.868,159.906
C03158=1017.576,316.301,-142.907,170.287,50.864,159.906
C03159=1017.581,316.548,-142.941,170.294,50.860,159.906
C03160=1017.588,316.795,-142.974,170.300,50.856,159.906
C03161=1017.595,317.044,-143.007,170.306,50.852,159.907
C03162=1017.602,317.291,-143.041,170.313,50.848,159.907
C03163=1017.608,317.539,-143.074,170.319,50.844,159.907
C03164=1017.614,317.786,-143.108,170.325,50.840,159.907
C03165=1017.621,318.035,-143.141,170.332,50.836,159.907
C03166=1017.628,318.281,-143.175,170.338,50.833,159.907
C03167=1017.635,318.529,-143.208,170.344,50.829,159.908
C03168=1017.641,318.777,-143.242,170.350,50.825,159.908
C03169=1017.648,319.025,-143.276,170.356,50.821,159.908
C03170=1017.654,319.272,-143.308,170.363,50.818,159.908
C03171=1017.661,319.520,-143.342,170.369,50.814,159.909
C03172=1017.668,319.768,-143.376,170.375,50.810,159.909
C03173=1017.674,320.015,-143.410,170.382,50.806,159.909
C03174=1017.681,320.263,-143.443,170.389,50.802,159.909
C03175=1017.688,320.510,-143.477,170.395,50.798,159.909
C03176=1017.695,320.758,-143.510,170.401,50.795,159.910
C03177=1017.701,321.006,-143.545,170.407,50.791,159.910
C03178=1017.708,321.253,-143.578,170.414,50.787,159.910
C03179=1017.715,321.501,-143.611,170.420,50.783,159.910
C03180=1017.722,321.749,-143.645,170.426,50.780,159.910
C03181=1017.728,321.996,-143.679,170.433,50.776,159.911
C03182=1017.736,322.258,-143.714,170.439,50.772,159.911
C03183=1017.743,322.521,-143.751,170.447,50.768,159.911
C03184=1017.750,322.783,-143.787,170.453,50.764,159.911
C03185=1017.757,323.046,-143.823,170.460,50.760,159.912
C03186=1017.764,323.293,-143.856,170.467,50.757,159.912
C03187=1017.771,323.540,-143.890,170.473,50.753,159.912
C03188=1017.778,323.788,-143.924,170.479,50.749,159.913
C03189=1017.785,324.036,-143.958,170.485,50.745,159.913
C03190=1017.792,324.284,-143.992,170.493,50.741,159.913
C03191=1017.799,324.531,-144.026,170.499,50.738,159.913
C03192=1017.806,324.778,-144.059,170.506,50.734,159.914
C03193=1017.812,325.026,-144.094,170.512,50.731,159.914
C03194=1017.819,325.274,-144.127,170.518,50.728,159.914
C03195=1017.827,325.522,-144.161,170.525,50.724,159.914
C03196=1017.833,325.769,-144.196,170.532,50.720,159.915
C03197=1017.841,326.017,-144.230,170.539,50.717,159.915
C03198=1017.848,326.264,-144.264,170.545,50.713,159.915
C03199=1017.854,326.512,-144.298,170.551,50.710,159.916
C03200=1017.861,326.759,-144.333,170.558,50.706,159.916
C03201=1017.868,327.007,-144.367,170.564,50.703,159.916
C03202=1017.874,327.254,-144.402,170.570,50.699,159.917
C03203=1017.882,327.502,-144.436,170.578,50.696,159.917
C03204=1017.888,327.749,-144.471,170.585,50.693,159.918
C03205=1017.895,327.997,-144.506,170.591,50.689,159.918
C03206=1017.902,328.244,-144.541,170.598,50.686,159.918
C03207=1017.909,328.492,-144.575,170.604,50.683,159.919
C03208=1017.916,328.739,-144.610,170.610,50.679,159.919
C03209=1017.921,328.987,-144.644,170.617,50.676,159.919
C03210=1017.929,329.234,-144.678,170.625,50.672,159.920
C03211=1017.936,329.481,-144.713,170.631,50.669,159.920
C03212=1017.942,329.729,-144.748,170.638,50.666,159.920
C03213=1017.950,329.976,-144.782,170.644,50.662,159.921
C03214=1017.956,330.223,-144.817,170.651,50.659,159.921
C03215=1017.963,330.472,-144.852,170.657,50.656,159.922
C03216=1017.970,330.720,-144.887,170.664,50.652,159.922
C03217=1017.978,330.967,-144.922,170.671,50.649,159.922
C03218=1017.984,331.214,-144.957,170.678,50.646,159.923
C03219=1017.991,331.462,-144.991,170.685,50.643,159.923
C03220=1017.998,331.709,-145.026,170.691,50.640,159.923
C03221=1018.005,331.956,-145.061,170.698,50.637,159.924
C03222=1018.012,332.204,-145.096,170.705,50.633,159.924
C03223=1018.020,332.451,-145.131,170.712,50.630,159.925
C03224=1018.026,332.698,-145.166,170.719,50.627,159.925
C03225=1018.034,332.946,-145.201,170.725,50.624,159.926
C03226=1018.040,333.194,-145.237,170.732,50.621,159.926
C03227=1018.047,333.441,-145.272,170.739,50.618,159.926
C03228=1018.054,333.688,-145.307,170.746,50.614,159.927
C03229=1018.061,333.936,-145.342,170.753,50.611,159.927
C03230=1018.067,334.183,-145.377,170.759,50.608,159.928
C03231=1018.075,334.431,-145.413,170.766,50.605,159.928
C03232=1018.082,334.678,-145.448,170.773,50.602,159.928
C03233=1018.088,334.926,-145.483,170.780,50.599,159.929
C03234=1018.095,335.173,-145.519,170.787,50.596,159.930
C03235=1018.103,335.421,-145.554,170.794,50.593,159.930
C03236=1018.110,335.668,-145.589,170.801,50.590,159.930
C03237=1018.116,335.915,-145.625,170.808,50.587,159.931
C03238=1018.123,336.162,-145.660,170.814,50.584,159.931
C03239=1018.131,336.410,-145.696,170.822,50.581,159.932
C03240=1018.138,336.658,-145.731,170.828,50.578,159.932
C03241=1018.144,336.905,-145.766,170.835,50.575,159.933
C03242=1018.152,337.163,-145.803,170.843,50.572,159.933
C03243=1018.160,337.421,-145.841,170.850,50.569,159.934
C03244=1018.167,337.679,-145.878,170.858,50.566,159.935
C03245=1018.174,337.937,-145.915,170.864,50.563,159.935
C03246=1018.182,338.185,-145.950,170.871,50.560,159.935
C03247=1018.189,338.432,-145.986,170.879,50.557,159.936
C03248=1018.196,338.679,-146.021,170.886,50.554,159.936
C03249=1018.203,338.926,-146.057,170.893,50.551,159.937
C03250=1018.210,339.174,-146.093,170.899,50.548,159.937
C03251=1018.218,339.421,-146.129,170.907,50.545,159.938
C03252=1018.225,339.668,-146.165,170.914,50.542,159.939
C03253=1018.232,339.916,-146.200,170.921,50.540,159.939
C03254=1018.239,340.163,-146.237,170.928,50.537,159.940
C03255=1018.246,340.411,-146.273,170.936,50.534,159.940
C03256=1018.253,340.657,-146.309,170.943,50.532,159.941
C03257=1018.261,340.905,-146.344,170.950,50.529,159.941
C03258=1018.268,341.152,-146.380,170.956,50.526,159.942
C03259=1018.275,341.400,-146.417,170.964,50.523,159.943
C03260=1018.282,341.647,-146.453,170.971,50.521,159.943
C03261=1018.289,341.894,-146.489,170.978,50.518,159.944
C03262=1018.296,342.141,-146.525,170.985,50.515,159.944
C03263=1018.303,342.389,-146.561,170.993,50.512,159.945
C03264=1018.311,342.637,-146.597,171.000,50.510,159.945
C03265=1018.318,342.883,-146.633,171.007,50.508,159.946
C03266=1018.326,343.131,-146.669,171.015,50.505,159.947
C03267=1018.332,343.378,-146.706,171.022,50.502,159.947
C03268=1018.340,343.625,-146.742,171.029,50.499,159.948
C03269=1018.348,343.872,-146.779,171.036,50.497,159.948
C03270=1018.354,344.119,-146.815,171.044,50.494,159.949
C03271=1018.362,344.367,-146.851,171.051,50.491,159.950
C03272=1018.369,344.614,-146.888,171.058,50.489,159.950
C03273=1018.376,344.861,-146.924,171.066,50.486,159.951
C03274=1018.383,345.109,-146.960,171.073,50.484,159.952
C03275=1018.391,345.356,-146.996,171.080,50.481,159.952
C03276=1018.398,345.603,-147.034,171.088,50.479,159.953
C03277=1018.405,345.850,-147.070,171.095,50.476,159.953
C03278=1018.413,346.097,-147.106,171.102,50.474,159.954
C03279=1018.420,346.345,-147.143,171.110,50.471,159.955
C03280=1018.428,346.592,-147.180,171.117,50.469,159.956
C03281=1018.436,346.839,-147.216,171.124,50.467,159.956
C03282=1018.442,347.087,-147.253,171.132,50.464,159.957
C03283=1018.450,347.333,-147.289,171.139,50.461,159.957
C03284=1018.457,347.581,-147.326,171.147,50.459,159.958
C03285=1018.465,347.828,-147.363,171.155,50.457,159.959
C03286=1018.472,348.076,-147.400,171.162,50.454,159.960
C03287=1018.480,348.322,-147.437,171.170,50.451,159.960
C03288=1018.487,348.570,-147.474,171.177,50.450,159.961
C03289=1018.494,348.816,-147.510,171.184,50.447,159.962
C03290=1018.501,349.063,-147.548,171.192,50.445,159.963
C03291=1018.509,349.310,-147.585,171.199,50.443,159.963
C03292=1018.516,349.558,-147.622,171.206,50.440,159.964
C03293=1018.523,349.805,-147.659,171.215,50.438,159.965
C03294=1018.531,350.052,-147.696,171.222,50.435,159.965
C03295=1018.538,350.300,-147.733,171.230,50.433,159.966
C03296=1018.546,350.547,-147.770,171.237,50.431,159.967
C03297=1018.554,350.794,-147.807,171.245,50.429,159.968
C03298=1018.561,351.041,-147.845,171.253,50.426,159.968
C03299=1018.569,351.288,-147.882,171.260,50.424,159.969
C03300=1018.576,351.535,-147.919,171.268,50.422,159.970
C03301=1018.584,351.782,-147.955,171.275,50.420,159.971
C03302=1018.592,352.038,-147.994,171.284,50.418,159.972
C03303=1018.599,352.293,-148.033,171.291,50.415,159.972
C03304=1018.608,352.548,-148.072,171.299,50.413,159.973
C03305=1018.616,352.804,-148.111,171.308,50.411,159.974
C03306=1018.623,353.051,-148.148,171.315,50.409,159.975
C03307=1018.631,353.297,-148.185,171.323,50.406,159.975
C03308=1018.638,353.545,-148.223,171.331,50.404,159.976
C03309=1018.645,353.792,-148.260,171.339,50.402,159.977
C03310=1018.653,354.039,-148.297,171.346,50.400,159.978
C03311=1018.661,354.286,-148.335,171.354,50.398,159.979
C03312=1018.669,354.534,-148.372,171.362,50.396,159.979
C03313=1018.676,354.780,-148.411,171.370,50.394,159.980
C03314=1018.684,355.027,-148.448,171.378,50.392,159.981
C03315=1018.691,355.274,-148.485,171.386,50.390,159.982
C03316=1018.699,355.521,-148.524,171.393,50.388,159.983
C03317=1018.707,355.768,-148.561,171.402,50.386,159.984
C03318=1018.714,356.016,-148.599,171.409,50.384,159.985
C03319=1018.722,356.262,-148.636,171.417,50.382,159.985
C03320=1018.730,356.510,-148.674,171.425,50.380,159.986
C03321=1018.738,356.756,-148.713,171.433,50.378,159.987
C03322=1018.745,357.003,-148.750,171.441,50.376,159.988
C03323=1018.754,357.250,-148.788,171.449,50.374,159.989
C03324=1018.761,357.497,-148.826,171.456,50.372,159.990
C03325=1018.769,357.744,-148.864,171.465,50.370,159.991
C03326=1018.776,357.992,-148.902,171.473,50.368,159.992
C03327=1018.784,358.238,-148.940,171.481,50.366,159.992
C03328=1018.792,358.485,-148.979,171.488,50.364,159.993
C03329=1018.800,358.732,-149.016,171.497,50.362,159.994
C03330=1018.808,358.979,-149.054,171.506,50.361,159.995
C03331=1018.816,359.226,-149.092,171.513,50.359,159.996
C03332=1018.824,359.473,-149.131,171.521,50.357,159.997
C03333=1018.831,359.720,-149.169,171.529,50.355,159.998
C03334=1018.839,359.967,-149.207,171.538,50.353,159.999
C03335=1018.847,360.214,-149.245,171.545,50.352,160.000
C03336=1018.854,360.461,-149.284,171.554,50.350,160.001
C03337=1018.862,360.708,-149.323,171.563,50.348,160.002
C03338=1018.869,360.955,-149.361,171.570,50.346,160.003
C03339=1018.878,361.202,-149.400,171.579,50.345,160.004
C03340=1018.886,361.449,-149.438,171.586,50.343,160.005
C03341=1018.894,361.695,-149.477,171.595,50.342,160.006
C03342=1018.902,361.942,-149.516,171.603,50.339,160.007
C03343=1018.909,362.189,-149.554,171.611,50.338,160.008
C03344=1018.917,362.436,-149.593,171.620,50.337,160.009
C03345=1018.926,362.683,-149.631,171.628,50.334,160.010
C03346=1018.932,362.930,-149.670,171.636,50.333,160.011
C03347=1018.941,363.176,-149.710,171.645,50.332,160.012
C03348=1018.949,363.424,-149.748,171.653,50.329,160.013
C03349=1018.957,363.670,-149.786,171.661,50.328,160.014
C03350=1018.965,363.917,-149.826,171.670,50.327,160.015
C03351=1018.973,364.164,-149.864,171.679,50.325,160.016
C03352=1018.981,364.410,-149.903,171.686,50.323,160.017
C03353=1018.989,364.657,-149.942,171.695,50.322,160.018
C03354=1018.997,364.904,-149.980,171.703,50.320,160.019
C03355=1019.005,365.151,-150.020,171.712,50.319,160.020
C03356=1019.013,365.398,-150.059,171.720,50.317,160.021
C03357=1019.021,365.644,-150.098,171.729,50.316,160.022
C03358=1019.029,365.892,-150.137,171.738,50.314,160.023
C03359=1019.038,366.138,-150.176,171.746,50.313,160.024
C03360=1019.046,366.385,-150.215,171.754,50.312,160.025
C03361=1019.054,366.632,-150.254,171.763,50.310,160.026
C03362=1019.062,366.895,-150.295,171.772,50.308,160.027
C03363=1019.071,367.158,-150.337,171.781,50.306,160.029
C03364=1019.081,367.420,-150.379,171.790,50.305,160.030
C03365=1019.089,367.683,-150.420,171.799,50.304,160.031
C03366=1019.097,367.930,-150.460,171.808,50.302,160.032
C03367=1019.105,368.177,-150.499,171.817,50.301,160.033
C03368=1019.113,368.424,-150.539,171.826,50.299,160.034
C03369=1019.121,368.670,-150.579,171.834,50.299,160.035
C03370=1019.129,368.917,-150.618,171.843,50.297,160.037
C03371=1019.138,369.164,-150.658,171.851,50.296,160.038
C03372=1019.145,369.411,-150.698,171.861,50.295,160.039
C03373=1019.154,369.657,-150.737,171.869,50.293,160.040
C03374=1019.162,369.904,-150.776,171.878,50.291,160.041
C03375=1019.170,370.151,-150.816,171.886,50.291,160.042
C03376=1019.179,370.397,-150.856,171.895,50.289,160.043
C03377=1019.186,370.644,-150.896,171.904,50.288,160.045
C03378=1019.195,370.890,-150.936,171.913,50.287,160.046
C03379=1019.203,371.137,-150.975,171.922,50.286,160.047
C03380=1019.212,371.384,-151.016,171.931,50.284,160.048
C03381=1019.220,371.631,-151.056,171.940,50.283,160.050
C03382=1019.228,371.877,-151.095,171.949,50.282,160.051
C03383=1019.237,372.123,-151.135,171.957,50.281,160.052
C03384=1019.245,372.370,-151.175,171.966,50.280,160.053
C03385=1019.253,372.617,-151.214,171.975,50.279,160.054
C03386=1019.262,372.864,-151.255,171.984,50.278,160.056
C03387=1019.270,373.110,-151.295,171.993,50.277,160.057
C03388=1019.278,373.357,-151.335,172.003,50.276,160.058
C03389=1019.287,373.604,-151.375,172.011,50.274,160.059
C03390=1019.295,373.850,-151.416,172.020,50.273,160.061
C03391=1019.304,374.097,-151.455,172.030,50.272,160.062
C03392=1019.313,374.343,-151.495,172.039,50.271,160.063
C03393=1019.321,374.590,-151.536,172.048,50.270,160.064
C03394=1019.330,374.836,-151.575,172.057,50.269,160.066
C03395=1019.338,375.083,-151.616,172.066,50.268,160.067
C03396=1019.347,375.329,-151.656,172.075,50.267,160.068
C03397=1019.356,375.576,-151.697,172.084,50.266,160.069
C03398=1019.364,375.823,-151.737,172.093,50.265,160.071
C03399=1019.372,376.069,-151.777,172.103,50.264,160.072
C03400=1019.381,376.316,-151.818,172.113,50.263,160.074
C03401=1019.390,376.562,-151.858,172.122,50.262,160.075
C03402=1019.398,376.809,-151.899,172.131,50.261,160.076
C03403=1019.406,377.055,-151.940,172.140,50.260,160.078
C03404=1019.415,377.302,-151.981,172.150,50.259,160.079
C03405=1019.423,377.548,-152.022,172.159,50.259,160.080
C03406=1019.433,377.795,-152.063,172.168,50.258,160.082
C03407=1019.441,378.041,-152.103,172.178,50.257,160.083
C03408=1019.449,378.288,-152.144,172.187,50.256,160.084
C03409=1019.457,378.534,-152.185,172.196,50.256,160.086
C03410=1019.466,378.781,-152.227,172.205,50.255,160.087
C03411=1019.475,379.027,-152.267,172.216,50.254,160.089
C03412=1019.484,379.274,-152.308,172.225,50.253,160.090
C03413=1019.492,379.520,-152.350,172.234,50.252,160.091
C03414=1019.500,379.766,-152.390,172.244,50.252,160.093
C03415=1019.510,380.012,-152.431,172.253,50.251,160.094
C03416=1019.519,380.259,-152.472,172.262,50.250,160.096
C03417=1019.527,380.505,-152.514,172.273,50.250,160.097
C03418=1019.536,380.752,-152.555,172.282,50.249,160.099
C03419=1019.545,380.998,-152.596,172.292,50.248,160.100
C03420=1019.554,381.245,-152.637,172.301,50.247,160.101
C03421=1019.563,381.491,-152.678,172.311,50.247,160.103
C03422=1019.573,381.776,-152.726,172.322,50.246,160.105
C03423=1019.583,382.061,-152.774,172.334,50.245,160.106
C03424=1019.593,382.346,-152.822,172.344,50.245,160.108
C03425=1019.604,382.631,-152.869,172.356,50.244,160.110
C03426=1019.613,382.877,-152.911,172.365,50.243,160.111
C03427=1019.622,383.124,-152.953,172.376,50.242,160.113
C03428=1019.631,383.371,-152.994,172.386,50.242,160.114
C03429=1019.639,383.617,-153.035,172.395,50.242,160.116
C03430=1019.649,383.863,-153.076,172.406,50.241,160.117
C03431=1019.658,384.109,-153.118,172.415,50.241,160.119
C03432=1019.667,384.355,-153.160,172.425,50.240,160.121
C03433=1019.675,384.602,-153.201,172.435,50.239,160.122
C03434=1019.685,384.849,-153.244,172.445,50.239,160.124
C03435=1019.695,385.095,-153.285,172.455,50.238,160.125
C03436=1019.704,385.341,-153.326,172.465,50.238,160.127
C03437=1019.713,385.587,-153.369,172.474,50.238,160.128
C03438=1019.722,385.833,-153.411,172.485,50.237,160.130
C03439=1019.731,386.080,-153.452,172.495,50.237,160.132
C03440=1019.740,386.326,-153.494,172.505,50.236,160.133
C03441=1019.748,386.572,-153.537,172.515,50.236,160.135
C03442=1019.757,386.818,-153.579,172.525,50.235,160.136
C03443=1019.766,387.064,-153.621,172.535,50.235,160.138
C03444=1019.776,387.311,-153.663,172.546,50.235,160.140
C03445=1019.785,387.557,-153.706,172.556,50.235,160.141
C03446=1019.794,387.803,-153.747,172.566,50.234,160.143
C03447=1019.803,388.049,-153.790,172.576,50.234,160.145
C03448=1019.813,388.296,-153.832,172.587,50.234,160.146
C03449=1019.822,388.542,-153.874,172.597,50.234,160.148
C03450=1019.831,388.788,-153.917,172.607,50.233,160.150
C03451=1019.840,389.034,-153.960,172.617,50.233,160.151
C03452=1019.849,389.281,-154.002,172.628,50.233,160.153
C03453=1019.859,389.526,-154.044,172.638,50.233,160.155
C03454=1019.868,389.772,-154.087,172.649,50.232,160.156
C03455=1019.878,390.019,-154.129,172.660,50.232,160.158
C03456=1019.886,390.265,-154.173,172.669,50.232,160.160
C03457=1019.896,390.511,-154.215,172.680,50.232,160.161
C03458=1019.905,390.757,-154.258,172.691,50.232,160.163
C03459=1019.914,391.003,-154.300,172.701,50.232,160.165
C03460=1019.924,391.249,-154.343,172.712,50.232,160.167
C03461=1019.933,391.495,-154.386,172.723,50.231,160.169
C03462=1019.943,391.742,-154.429,172.733,50.232,160.170
C03463=1019.952,391.987,-154.471,172.744,50.231,160.172
C03464=1019.962,392.234,-154.514,172.754,50.231,160.174
C03465=1019.972,392.480,-154.558,172.764,50.231,160.176
C03466=1019.980,392.726,-154.601,172.775,50.231,160.177
C03467=1019.990,392.972,-154.643,172.786,50.231,160.179
C03468=1019.999,393.218,-154.687,172.797,50.231,160.181
C03469=1020.009,393.464,-154.730,172.807,50.231,160.183
C03470=1020.018,393.709,-154.773,172.818,50.232,160.185
C03471=1020.028,393.956,-154.816,172.829,50.231,160.187
C03472=1020.038,394.202,-154.860,172.840,50.231,160.188
C03473=1020.047,394.447,-154.902,172.852,50.232,160.190
C03474=1020.056,394.694,-154.947,172.861,50.232,160.192
C03475=1020.066,394.939,-154.990,172.872,50.232,160.194
C03476=1020.076,395.186,-155.033,172.884,50.232,160.196
C03477=1020.085,395.431,-155.077,172.895,50.232,160.198
C03478=1020.095,395.677,-155.120,172.906,50.232,160.200
C03479=1020.105,395.923,-155.164,172.917,50.232,160.202
C03480=1020.115,396.170,-155.207,172.928,50.232,160.204
C03481=1020.124,396.416,-155.251,172.939,50.232,160.205
C03482=1020.137,396.738,-155.308,172.953,50.233,160.208
C03483=1020.150,397.060,-155.365,172.968,50.233,160.211
C03484=1020.162,397.383,-155.423,172.983,50.234,160.213
C03485=1020.176,397.705,-155.480,172.998,50.234,160.216
C03486=1020.185,397.951,-155.525,173.009,50.234,160.218
C03487=1020.196,398.197,-155.568,173.020,50.234,160.220
C03488=1020.205,398.443,-155.612,173.032,50.235,160.222
C03489=1020.215,398.689,-155.657,173.043,50.235,160.224
C03490=1020.225,398.935,-155.700,173.054,50.235,160.226
C03491=1020.234,399.181,-155.745,173.065,50.236,160.228
C03492=1020.245,399.426,-155.789,173.077,50.236,160.230
C03493=1020.254,399.672,-155.833,173.088,50.237,160.232
C03494=1020.264,399.918,-155.878,173.099,50.237,160.234
C03495=1020.274,400.163,-155.921,173.112,50.237,160.236
C03496=1020.284,400.409,-155.966,173.123,50.237,160.238
C03497=1020.294,400.655,-156.010,173.134,50.238,160.240
C03498=1020.304,400.901,-156.055,173.146,50.239,160.242
C03499=1020.314,401.146,-156.100,173.157,50.239,160.244
C03500=1020.323,401.393,-156.144,173.169,50.240,160.246
C03501=1020.333,401.638,-156.189,173.181,50.240,160.249
C03502=1020.343,401.883,-156.233,173.193,50.240,160.251
C03503=1020.354,402.130,-156.278,173.204,50.241,160.253
C03504=1020.363,402.375,-156.323,173.216,50.242,160.255
C03505=1020.373,402.621,-156.368,173.228,50.242,160.257
C03506=1020.384,402.866,-156.412,173.240,50.243,160.259
C03507=1020.394,403.112,-156.457,173.251,50.244,160.262
C03508=1020.404,403.357,-156.502,173.263,50.244,160.264
C03509=1020.414,403.604,-156.547,173.275,50.245,160.266
C03510=1020.424,403.849,-156.592,173.287,50.246,160.268
C03511=1020.435,404.095,-156.636,173.299,50.246,160.270
C03512=1020.445,404.340,-156.682,173.311,50.247,160.272
C03513=1020.455,404.586,-156.727,173.323,50.247,160.275
C03514=1020.465,404.832,-156.772,173.335,50.248,160.277
C03515=1020.475,405.077,-156.818,173.347,50.249,160.279
C03516=1020.486,405.323,-156.862,173.360,50.250,160.282
C03517=1020.496,405.569,-156.907,173.371,50.251,160.284
C03518=1020.507,405.814,-156.953,173.384,50.251,160.286
C03519=1020.517,406.060,-156.998,173.396,50.252,160.288
C03520=1020.527,406.305,-157.044,173.409,50.253,160.291
C03521=1020.538,406.551,-157.089,173.420,50.253,160.293
C03522=1020.549,406.797,-157.134,173.433,50.254,160.295
C03523=1020.559,407.042,-157.180,173.445,50.255,160.297
C03524=1020.569,407.288,-157.225,173.457,50.256,160.300
C03525=1020.581,407.533,-157.271,173.470,50.256,160.302
C03526=1020.591,407.779,-157.316,173.482,50.258,160.305
C03527=1020.602,408.025,-157.362,173.495,50.258,160.307
C03528=1020.612,408.270,-157.407,173.507,50.259,160.309
C03529=1020.622,408.516,-157.453,173.520,50.260,160.312
C03530=1020.634,408.761,-157.498,173.532,50.261,160.314
C03531=1020.644,409.007,-157.544,173.545,50.262,160.316
C03532=1020.655,409.252,-157.590,173.557,50.263,160.319
C03533=1020.665,409.498,-157.637,173.570,50.264,160.321
C03534=1020.675,409.744,-157.683,173.583,50.264,160.324
C03535=1020.686,409.989,-157.729,173.596,50.266,160.326
C03536=1020.697,410.234,-157.775,173.608,50.267,160.329
C03537=1020.707,410.480,-157.821,173.621,50.268,160.331
C03538=1020.718,410.725,-157.868,173.634,50.269,160.333
C03539=1020.730,410.971,-157.914,173.647,50.270,160.336
C03540=1020.740,411.217,-157.960,173.660,50.271,160.338
C03541=1020.751,411.462,-158.006,173.673,50.272,160.341
C03542=1020.766,411.807,-158.072,173.690,50.274,160.344
C03543=1020.781,412.153,-158.137,173.709,50.276,160.348
C03544=1020.797,412.498,-158.202,173.727,50.277,160.352
C03545=1020.811,412.843,-158.268,173.746,50.278,160.355
C03546=1020.823,413.088,-158.315,173.760,50.280,160.358
C03547=1020.834,413.333,-158.362,173.773,50.281,160.361
C03548=1020.845,413.579,-158.408,173.786,50.282,160.363
C03549=1020.856,413.824,-158.455,173.799,50.283,160.366
C03550=1020.867,414.069,-158.502,173.812,50.285,160.368
C03551=1020.878,414.316,-158.549,173.826,50.286,160.371
C03552=1020.889,414.561,-158.595,173.839,50.287,160.374
C03553=1020.901,414.806,-158.643,173.852,50.289,160.376
C03554=1020.912,415.051,-158.690,173.866,50.290,160.379
C03555=1020.923,415.296,-158.737,173.880,50.291,160.382
C03556=1020.934,415.542,-158.784,173.893,50.293,160.384
C03557=1020.945,415.787,-158.831,173.907,50.294,160.387
C03558=1020.956,416.033,-158.879,173.920,50.295,160.390
C03559=1020.967,416.278,-158.926,173.933,50.297,160.392
C03560=1020.979,416.523,-158.973,173.948,50.298,160.395
C03561=1020.989,416.769,-159.021,173.961,50.300,160.398
C03562=1021.001,417.013,-159.068,173.975,50.301,160.401
C03563=1021.012,417.259,-159.115,173.989,50.303,160.404
C03564=1021.023,417.504,-159.164,174.003,50.304,160.406
C03565=1021.035,417.749,-159.211,174.016,50.306,160.409
C03566=1021.045,417.994,-159.258,174.030,50.307,160.412
C03567=1021.057,418.239,-159.306,174.044,50.309,160.415
